REGION Network 17: AGAIN OFF TIME START AFTER RECIRCULATION OVER
   RUNG wire#powerrail
      Contact( "AlwaysTRUE" )
      { S7_Templates := "SrcType := Int" } EQ_Contact(in1 := "MODE SELECTION DB"."RO-2"."MODE BUFF", in2 := 1)
      { S7_Templates := "SrcType := Int" } EQ_Contact(in1 := "MODE SELECTION DB"."RO-2"."PROCESS BUFF", in2 := 2)
      { S7_Templates := "SrcType := Int" } EQ_Contact(in1 := "RO_2_LEVEL DB"."LEVEL HI RECIRC BUFF", in2 := 3)
      Contact( "TIMING_MIN_DB_10".DONE )
      Move(in := 4, out1 => "RO_2_LEVEL DB"."LEVEL HI RECIRC BUFF")
   END_RUNG
   // the same network as SCL:
   IF "AlwaysTRUE" AND ("MODE SELECTION DB"."RO-2"."MODE BUFF" = 1) AND ("MODE SELECTION DB"."RO-2"."PROCESS BUFF" = 2) AND ("RO_2_LEVEL DB"."LEVEL HI RECIRC BUFF" = 3) AND "TIMING_MIN_DB_10".DONE THEN
       "RO_2_LEVEL DB"."LEVEL HI RECIRC BUFF" := 4;
   END_IF;
END_REGION

REGION Network 18: AGAIN OFF TIME START AFTER RECIRCULATION OVER
   RUNG wire#powerrail
      Contact( "AlwaysTRUE" )
      { S7_Templates := "SrcType := Int" } EQ_Contact(in1 := "MODE SELECTION DB"."RO-2"."MODE BUFF", in2 := 1)
      { S7_Templates := "SrcType := Int" } EQ_Contact(in1 := "MODE SELECTION DB"."RO-2"."PROCESS BUFF", in2 := 2)
      { S7_Templates := "SrcType := Int" } EQ_Contact(in1 := "RO_2_LEVEL DB"."LEVEL HI RECIRC BUFF", in2 := 4)
      { S7_Templates := "time_type := Time" } "IEC_Timer_0_DB_95".TP(pt := T#2S, et =>)
      Move(in := 2, out1 => "RO_2_LEVEL DB"."LEVEL HI RECIRC BUFF")
   END_RUNG
   // the same network as SCL:
   "IEC_Timer_0_DB_95".TP(IN := "AlwaysTRUE" AND ("MODE SELECTION DB"."RO-2"."MODE BUFF" = 1) AND ("MODE SELECTION DB"."RO-2"."PROCESS BUFF" = 2) AND ("RO_2_LEVEL DB"."LEVEL HI RECIRC BUFF" = 4),
                          PT := T#2S);
   IF "IEC_Timer_0_DB_95".Q THEN "RO_2_LEVEL DB"."LEVEL HI RECIRC BUFF" := 2; END_IF;
END_REGION

REGION Network 19: REcirculation stop when level is normal
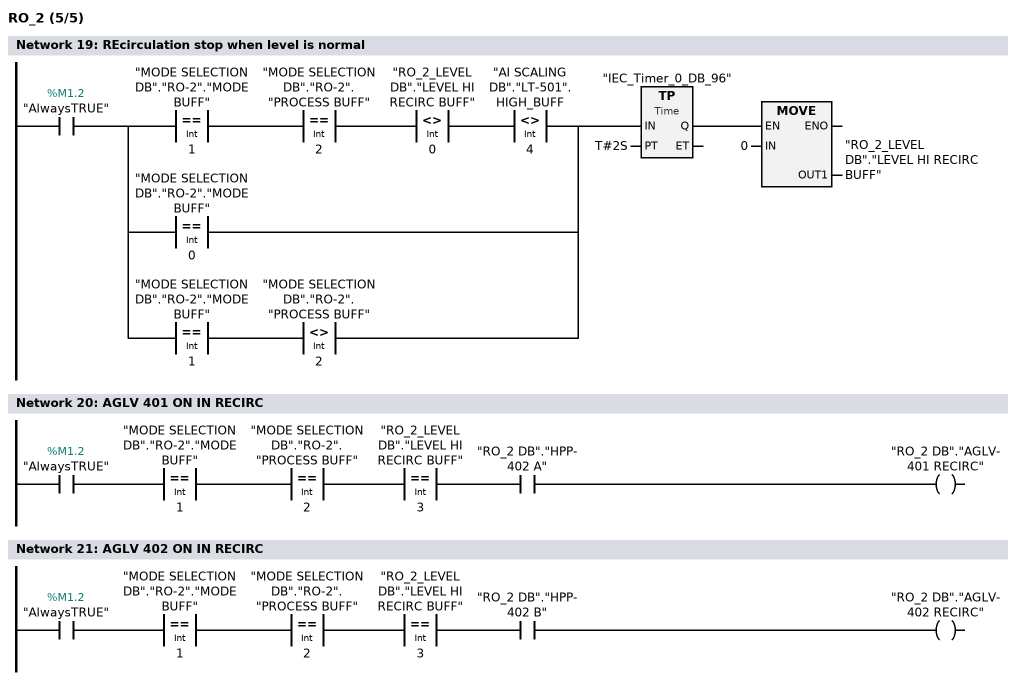
   RUNG wire#powerrail
      Contact( "AlwaysTRUE" )
      wire#w1
      { S7_Templates := "SrcType := Int" } EQ_Contact(in1 := "MODE SELECTION DB"."RO-2"."MODE BUFF", in2 := 1)
      { S7_Templates := "SrcType := Int" } EQ_Contact(in1 := "MODE SELECTION DB"."RO-2"."PROCESS BUFF", in2 := 2)
      { S7_Templates := "SrcType := Int" } NE_Contact(in1 := "RO_2_LEVEL DB"."LEVEL HI RECIRC BUFF", in2 := 0)
      { S7_Templates := "SrcType := Int" } NE_Contact(in1 := "AI SCALING DB"."LT-501".HIGH_BUFF, in2 := 4)
      wire#w2
      { S7_Templates := "time_type := Time" } "IEC_Timer_0_DB_96".TP(pt := T#2S, et =>)
      Move(in := 0, out1 => "RO_2_LEVEL DB"."LEVEL HI RECIRC BUFF")
   END_RUNG
   RUNG wire#w1
      { S7_Templates := "SrcType := Int" } EQ_Contact(in1 := "MODE SELECTION DB"."RO-2"."MODE BUFF", in2 := 0)
   END_RUNG wire#w2
   RUNG wire#w1
      { S7_Templates := "SrcType := Int" } EQ_Contact(in1 := "MODE SELECTION DB"."RO-2"."MODE BUFF", in2 := 1)
      { S7_Templates := "SrcType := Int" } NE_Contact(in1 := "MODE SELECTION DB"."RO-2"."PROCESS BUFF", in2 := 2)
   END_RUNG wire#w2
   // the same network as SCL:
   "IEC_Timer_0_DB_96".TP(IN := "AlwaysTRUE" AND ((("MODE SELECTION DB"."RO-2"."MODE BUFF" = 1) AND ("MODE SELECTION DB"."RO-2"."PROCESS BUFF" = 2) AND ("RO_2_LEVEL DB"."LEVEL HI RECIRC BUFF" <> 0) AND ("AI SCALING DB"."LT-501".HIGH_BUFF <> 4)) OR ("MODE SELECTION DB"."RO-2"."MODE BUFF" = 0) OR (("MODE SELECTION DB"."RO-2"."MODE BUFF" = 1) AND ("MODE SELECTION DB"."RO-2"."PROCESS BUFF" <> 2))),
                          PT := T#2S);
   IF "IEC_Timer_0_DB_96".Q THEN "RO_2_LEVEL DB"."LEVEL HI RECIRC BUFF" := 0; END_IF;
END_REGION

REGION Network 20: AGLV 401 ON IN RECIRC
   RUNG wire#powerrail
      Contact( "AlwaysTRUE" )
      { S7_Templates := "SrcType := Int" } EQ_Contact(in1 := "MODE SELECTION DB"."RO-2"."MODE BUFF", in2 := 1)
      { S7_Templates := "SrcType := Int" } EQ_Contact(in1 := "MODE SELECTION DB"."RO-2"."PROCESS BUFF", in2 := 2)
      { S7_Templates := "SrcType := Int" } EQ_Contact(in1 := "RO_2_LEVEL DB"."LEVEL HI RECIRC BUFF", in2 := 3)
      Contact( "RO_2 DB"."HPP-402 A" )
      Coil( "RO_2 DB"."AGLV-401 RECIRC" )
   END_RUNG
   // the same network as SCL:
   "RO_2 DB"."AGLV-401 RECIRC" := "AlwaysTRUE" AND ("MODE SELECTION DB"."RO-2"."MODE BUFF" = 1) AND ("MODE SELECTION DB"."RO-2"."PROCESS BUFF" = 2) AND ("RO_2_LEVEL DB"."LEVEL HI RECIRC BUFF" = 3) AND "RO_2 DB"."HPP-402 A";
END_REGION

REGION Network 21: AGLV 402 ON IN RECIRC
   RUNG wire#powerrail
      Contact( "AlwaysTRUE" )
      { S7_Templates := "SrcType := Int" } EQ_Contact(in1 := "MODE SELECTION DB"."RO-2"."MODE BUFF", in2 := 1)
      { S7_Templates := "SrcType := Int" } EQ_Contact(in1 := "MODE SELECTION DB"."RO-2"."PROCESS BUFF", in2 := 2)
      { S7_Templates := "SrcType := Int" } EQ_Contact(in1 := "RO_2_LEVEL DB"."LEVEL HI RECIRC BUFF", in2 := 3)
      Contact( "RO_2 DB"."HPP-402 B" )
      Coil( "RO_2 DB"."AGLV-402 RECIRC" )
   END_RUNG
   // the same network as SCL:
   "RO_2 DB"."AGLV-402 RECIRC" := "AlwaysTRUE" AND ("MODE SELECTION DB"."RO-2"."MODE BUFF" = 1) AND ("MODE SELECTION DB"."RO-2"."PROCESS BUFF" = 2) AND ("RO_2_LEVEL DB"."LEVEL HI RECIRC BUFF" = 3) AND "RO_2 DB"."HPP-402 B";
END_REGION
END_FUNCTION

FUNCTION "EDI" : Void   // FC12, LAD
{ S7_Optimized_Access := 'TRUE' }
// stored: SetENOAutomatically false
   VAR_TEMP   // added for the SCL form of the ladder/FBD networks
      _w1 : Bool;
   END_VAR
BEGIN

REGION Network 1: FEED PUMP
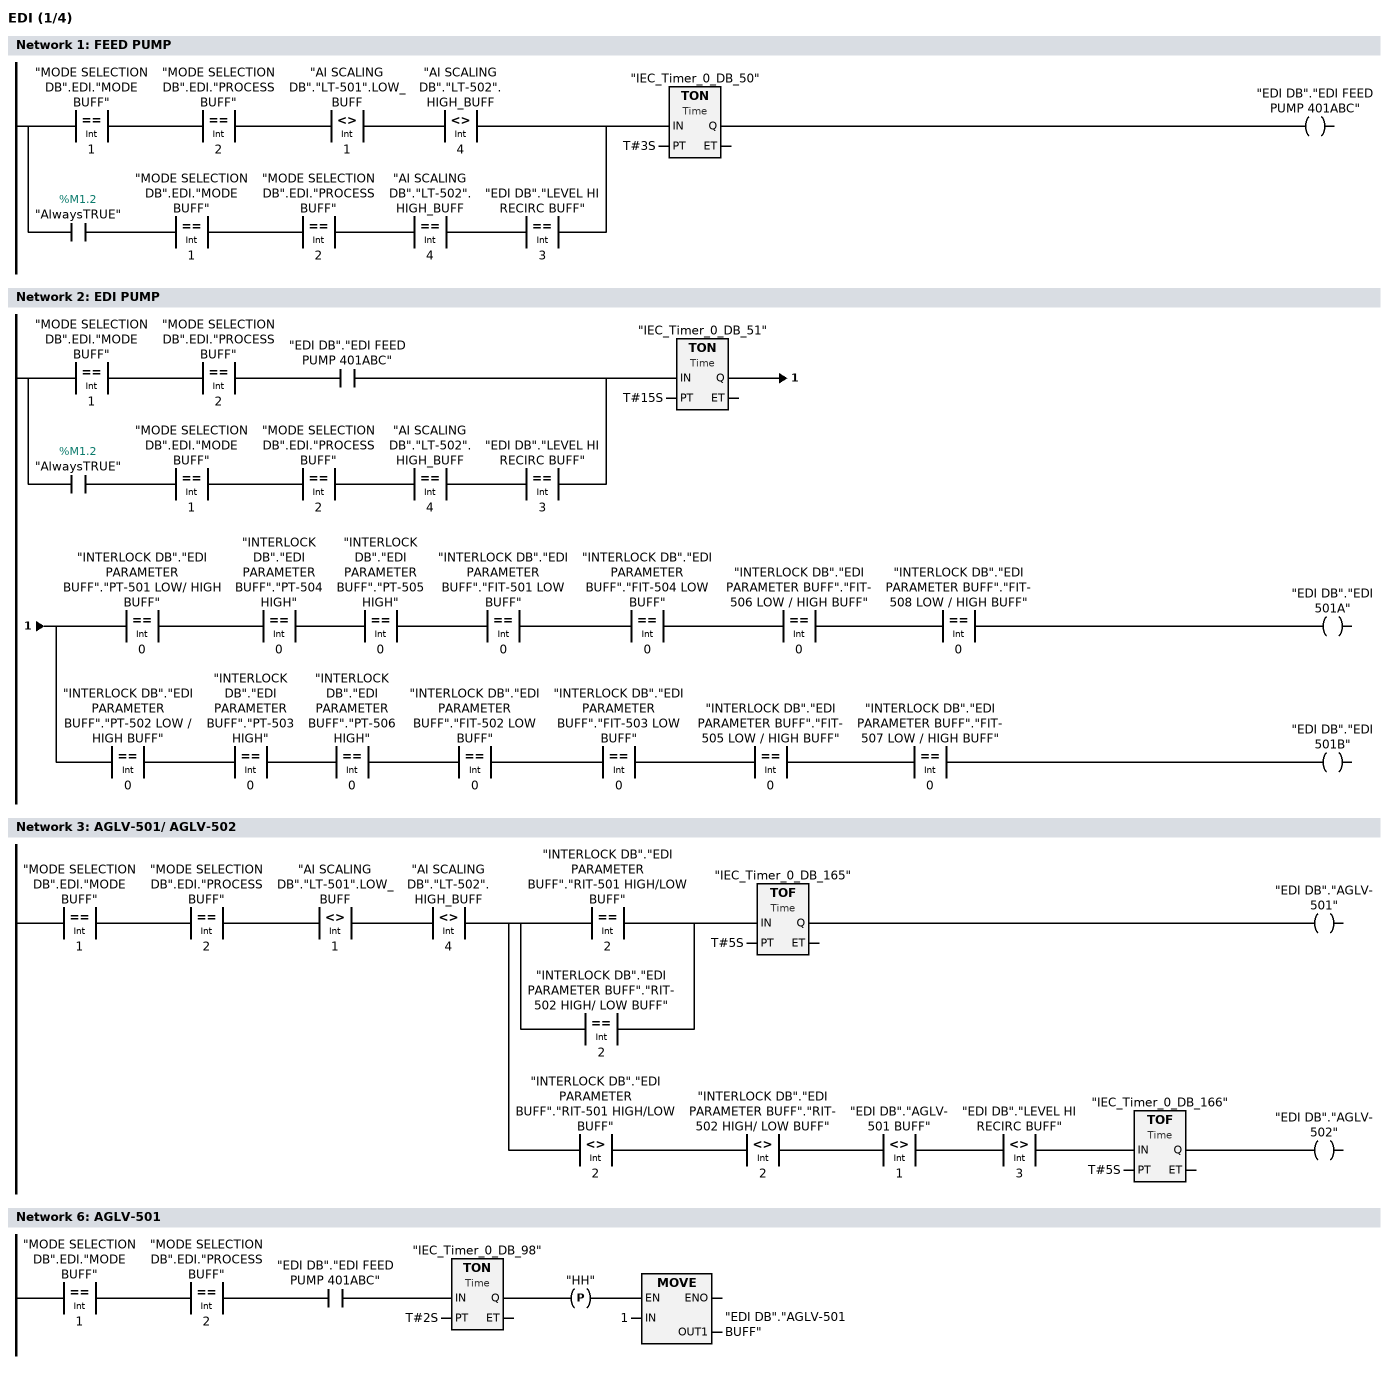
   RUNG wire#powerrail
      { S7_Templates := "SrcType := Int" } EQ_Contact(in1 := "MODE SELECTION DB".EDI."MODE BUFF", in2 := 1)
      { S7_Templates := "SrcType := Int" } EQ_Contact(in1 := "MODE SELECTION DB".EDI."PROCESS BUFF", in2 := 2)
      { S7_Templates := "SrcType := Int" } NE_Contact(in1 := "AI SCALING DB"."LT-501".LOW_BUFF, in2 := 1)
      { S7_Templates := "SrcType := Int" } NE_Contact(in1 := "AI SCALING DB"."LT-502".HIGH_BUFF, in2 := 4)
      wire#w1
      { S7_Templates := "time_type := Time" } "IEC_Timer_0_DB_50".TON(pt := T#3S, et =>)
      Coil( "EDI DB"."EDI FEED PUMP 401ABC" )
   END_RUNG
   RUNG wire#powerrail
      Contact( "AlwaysTRUE" )
      { S7_Templates := "SrcType := Int" } EQ_Contact(in1 := "MODE SELECTION DB".EDI."MODE BUFF", in2 := 1)
      { S7_Templates := "SrcType := Int" } EQ_Contact(in1 := "MODE SELECTION DB".EDI."PROCESS BUFF", in2 := 2)
      { S7_Templates := "SrcType := Int" } EQ_Contact(in1 := "AI SCALING DB"."LT-502".HIGH_BUFF, in2 := 4)
      { S7_Templates := "SrcType := Int" } EQ_Contact(in1 := "EDI DB"."LEVEL HI RECIRC BUFF", in2 := 3)
   END_RUNG wire#w1
   // the same network as SCL:
   "IEC_Timer_0_DB_50".TON(IN := (("MODE SELECTION DB".EDI."MODE BUFF" = 1) AND ("MODE SELECTION DB".EDI."PROCESS BUFF" = 2) AND ("AI SCALING DB"."LT-501".LOW_BUFF <> 1) AND ("AI SCALING DB"."LT-502".HIGH_BUFF <> 4)) OR ("AlwaysTRUE" AND ("MODE SELECTION DB".EDI."MODE BUFF" = 1) AND ("MODE SELECTION DB".EDI."PROCESS BUFF" = 2) AND ("AI SCALING DB"."LT-502".HIGH_BUFF = 4) AND ("EDI DB"."LEVEL HI RECIRC BUFF" = 3)),
                           PT := T#3S);
   "EDI DB"."EDI FEED PUMP 401ABC" := "IEC_Timer_0_DB_50".Q;
END_REGION

REGION Network 2: EDI PUMP
   RUNG wire#powerrail
      { S7_Templates := "SrcType := Int" } EQ_Contact(in1 := "MODE SELECTION DB".EDI."MODE BUFF", in2 := 1)
      { S7_Templates := "SrcType := Int" } EQ_Contact(in1 := "MODE SELECTION DB".EDI."PROCESS BUFF", in2 := 2)
      Contact( "EDI DB"."EDI FEED PUMP 401ABC" )
      wire#w1
      { S7_Templates := "time_type := Time" } "IEC_Timer_0_DB_51".TON(pt := T#15S, et =>)
      wire#w2
      { S7_Templates := "SrcType := Int" } EQ_Contact(in1 := "INTERLOCK DB"."EDI PARAMETER BUFF"."PT-501 LOW/ HIGH BUFF", in2 := 0)
      { S7_Templates := "SrcType := Int" } EQ_Contact(in1 := "INTERLOCK DB"."EDI PARAMETER BUFF"."PT-504 HIGH", in2 := 0)
      { S7_Templates := "SrcType := Int" } EQ_Contact(in1 := "INTERLOCK DB"."EDI PARAMETER BUFF"."PT-505 HIGH", in2 := 0)
      { S7_Templates := "SrcType := Int" } EQ_Contact(in1 := "INTERLOCK DB"."EDI PARAMETER BUFF"."FIT-501 LOW BUFF", in2 := 0)
      { S7_Templates := "SrcType := Int" } EQ_Contact(in1 := "INTERLOCK DB"."EDI PARAMETER BUFF"."FIT-504 LOW BUFF", in2 := 0)
      { S7_Templates := "SrcType := Int" } EQ_Contact(in1 := "INTERLOCK DB"."EDI PARAMETER BUFF"."FIT-506 LOW / HIGH BUFF", in2 := 0)
      { S7_Templates := "SrcType := Int" } EQ_Contact(in1 := "INTERLOCK DB"."EDI PARAMETER BUFF"."FIT-508 LOW / HIGH BUFF", in2 := 0)
      Coil( "EDI DB"."EDI 501A" )
   END_RUNG
   RUNG wire#powerrail
      Contact( "AlwaysTRUE" )
      { S7_Templates := "SrcType := Int" } EQ_Contact(in1 := "MODE SELECTION DB".EDI."MODE BUFF", in2 := 1)
      { S7_Templates := "SrcType := Int" } EQ_Contact(in1 := "MODE SELECTION DB".EDI."PROCESS BUFF", in2 := 2)
      { S7_Templates := "SrcType := Int" } EQ_Contact(in1 := "AI SCALING DB"."LT-502".HIGH_BUFF, in2 := 4)
      { S7_Templates := "SrcType := Int" } EQ_Contact(in1 := "EDI DB"."LEVEL HI RECIRC BUFF", in2 := 3)
   END_RUNG wire#w1
   RUNG wire#w2
      { S7_Templates := "SrcType := Int" } EQ_Contact(in1 := "INTERLOCK DB"."EDI PARAMETER BUFF"."PT-502 LOW / HIGH BUFF", in2 := 0)
      { S7_Templates := "SrcType := Int" } EQ_Contact(in1 := "INTERLOCK DB"."EDI PARAMETER BUFF"."PT-503 HIGH", in2 := 0)
      { S7_Templates := "SrcType := Int" } EQ_Contact(in1 := "INTERLOCK DB"."EDI PARAMETER BUFF"."PT-506 HIGH", in2 := 0)
      { S7_Templates := "SrcType := Int" } EQ_Contact(in1 := "INTERLOCK DB"."EDI PARAMETER BUFF"."FIT-502 LOW  BUFF", in2 := 0)
      { S7_Templates := "SrcType := Int" } EQ_Contact(in1 := "INTERLOCK DB"."EDI PARAMETER BUFF"."FIT-503 LOW BUFF", in2 := 0)
      { S7_Templates := "SrcType := Int" } EQ_Contact(in1 := "INTERLOCK DB"."EDI PARAMETER BUFF"."FIT-505 LOW / HIGH BUFF", in2 := 0)
      { S7_Templates := "SrcType := Int" } EQ_Contact(in1 := "INTERLOCK DB"."EDI PARAMETER BUFF"."FIT-507 LOW / HIGH BUFF", in2 := 0)
      Coil( "EDI DB"."EDI 501B" )
   END_RUNG
   // the same network as SCL:
   "IEC_Timer_0_DB_51".TON(IN := (("MODE SELECTION DB".EDI."MODE BUFF" = 1) AND ("MODE SELECTION DB".EDI."PROCESS BUFF" = 2) AND "EDI DB"."EDI FEED PUMP 401ABC") OR ("AlwaysTRUE" AND ("MODE SELECTION DB".EDI."MODE BUFF" = 1) AND ("MODE SELECTION DB".EDI."PROCESS BUFF" = 2) AND ("AI SCALING DB"."LT-502".HIGH_BUFF = 4) AND ("EDI DB"."LEVEL HI RECIRC BUFF" = 3)),
                           PT := T#15S);
   "EDI DB"."EDI 501A" := "IEC_Timer_0_DB_51".Q AND ("INTERLOCK DB"."EDI PARAMETER BUFF"."PT-501 LOW/ HIGH BUFF" = 0) AND ("INTERLOCK DB"."EDI PARAMETER BUFF"."PT-504 HIGH" = 0) AND ("INTERLOCK DB"."EDI PARAMETER BUFF"."PT-505 HIGH" = 0) AND ("INTERLOCK DB"."EDI PARAMETER BUFF"."FIT-501 LOW BUFF" = 0) AND ("INTERLOCK DB"."EDI PARAMETER BUFF"."FIT-504 LOW BUFF" = 0) AND ("INTERLOCK DB"."EDI PARAMETER BUFF"."FIT-506 LOW / HIGH BUFF" = 0) AND ("INTERLOCK DB"."EDI PARAMETER BUFF"."FIT-508 LOW / HIGH BUFF" = 0);
   "EDI DB"."EDI 501B" := "IEC_Timer_0_DB_51".Q AND ("INTERLOCK DB"."EDI PARAMETER BUFF"."PT-502 LOW / HIGH BUFF" = 0) AND ("INTERLOCK DB"."EDI PARAMETER BUFF"."PT-503 HIGH" = 0) AND ("INTERLOCK DB"."EDI PARAMETER BUFF"."PT-506 HIGH" = 0) AND ("INTERLOCK DB"."EDI PARAMETER BUFF"."FIT-502 LOW  BUFF" = 0) AND ("INTERLOCK DB"."EDI PARAMETER BUFF"."FIT-503 LOW BUFF" = 0) AND ("INTERLOCK DB"."EDI PARAMETER BUFF"."FIT-505 LOW / HIGH BUFF" = 0) AND ("INTERLOCK DB"."EDI PARAMETER BUFF"."FIT-507 LOW / HIGH BUFF" = 0);
END_REGION

REGION Network 3: AGLV-501/ AGLV-502
   RUNG wire#powerrail
      { S7_Templates := "SrcType := Int" } EQ_Contact(in1 := "MODE SELECTION DB".EDI."MODE BUFF", in2 := 1)
      { S7_Templates := "SrcType := Int" } EQ_Contact(in1 := "MODE SELECTION DB".EDI."PROCESS BUFF", in2 := 2)
      { S7_Templates := "SrcType := Int" } NE_Contact(in1 := "AI SCALING DB"."LT-501".LOW_BUFF, in2 := 1)
      { S7_Templates := "SrcType := Int" } NE_Contact(in1 := "AI SCALING DB"."LT-502".HIGH_BUFF, in2 := 4)
      wire#w1
      { S7_Templates := "SrcType := Int" } EQ_Contact(in1 := "INTERLOCK DB"."EDI PARAMETER BUFF"."RIT-501 HIGH/LOW BUFF", in2 := 2)
      wire#w2
      { S7_Templates := "time_type := Time" } "IEC_Timer_0_DB_165".TOF(pt := T#5S, et =>)
      Coil( "EDI DB"."AGLV-501" )
   END_RUNG
   RUNG wire#w1
      { S7_Templates := "SrcType := Int" } EQ_Contact(in1 := "INTERLOCK DB"."EDI PARAMETER BUFF"."RIT-502 HIGH/ LOW BUFF", in2 := 2)
   END_RUNG wire#w2
   RUNG wire#w1
      { S7_Templates := "SrcType := Int" } NE_Contact(in1 := "INTERLOCK DB"."EDI PARAMETER BUFF"."RIT-501 HIGH/LOW BUFF", in2 := 2)
      { S7_Templates := "SrcType := Int" } NE_Contact(in1 := "INTERLOCK DB"."EDI PARAMETER BUFF"."RIT-502 HIGH/ LOW BUFF", in2 := 2)
      { S7_Templates := "SrcType := Int" } NE_Contact(in1 := "EDI DB"."AGLV-501 BUFF", in2 := 1)
      { S7_Templates := "SrcType := Int" } NE_Contact(in1 := "EDI DB"."LEVEL HI RECIRC BUFF", in2 := 3)
      { S7_Templates := "time_type := Time" } "IEC_Timer_0_DB_166".TOF(pt := T#5S, et =>)
      Coil( "EDI DB"."AGLV-502" )
   END_RUNG
   // the same network as SCL:
   #_w1 := ("MODE SELECTION DB".EDI."MODE BUFF" = 1) AND ("MODE SELECTION DB".EDI."PROCESS BUFF" = 2) AND ("AI SCALING DB"."LT-501".LOW_BUFF <> 1) AND ("AI SCALING DB"."LT-502".HIGH_BUFF <> 4);
   "IEC_Timer_0_DB_165".TOF(IN := #_w1 AND (("INTERLOCK DB"."EDI PARAMETER BUFF"."RIT-501 HIGH/LOW BUFF" = 2) OR ("INTERLOCK DB"."EDI PARAMETER BUFF"."RIT-502 HIGH/ LOW BUFF" = 2)),
                           PT := T#5S);
   "EDI DB"."AGLV-501" := "IEC_Timer_0_DB_165".Q;
   "IEC_Timer_0_DB_166".TOF(IN := #_w1 AND ("INTERLOCK DB"."EDI PARAMETER BUFF"."RIT-501 HIGH/LOW BUFF" <> 2) AND ("INTERLOCK DB"."EDI PARAMETER BUFF"."RIT-502 HIGH/ LOW BUFF" <> 2) AND ("EDI DB"."AGLV-501 BUFF" <> 1) AND ("EDI DB"."LEVEL HI RECIRC BUFF" <> 3),
                           PT := T#5S);
   "EDI DB"."AGLV-502" := "IEC_Timer_0_DB_166".Q;
END_REGION

REGION Network 6: AGLV-501
   RUNG wire#powerrail
      { S7_Templates := "SrcType := Int" } EQ_Contact(in1 := "MODE SELECTION DB".EDI."MODE BUFF", in2 := 1)
      { S7_Templates := "SrcType := Int" } EQ_Contact(in1 := "MODE SELECTION DB".EDI."PROCESS BUFF", in2 := 2)
      Contact( "EDI DB"."EDI FEED PUMP 401ABC" )
      { S7_Templates := "time_type := Time" } "IEC_Timer_0_DB_98".TON(pt := T#2S, et =>)
      P_Trig( "HH" )
      Move(in := 1, out1 => "EDI DB"."AGLV-501 BUFF")
   END_RUNG
   // the same network as SCL:
   "IEC_Timer_0_DB_98".TON(IN := ("MODE SELECTION DB".EDI."MODE BUFF" = 1) AND ("MODE SELECTION DB".EDI."PROCESS BUFF" = 2) AND "EDI DB"."EDI FEED PUMP 401ABC",
                           PT := T#2S);
   #_w1 := "IEC_Timer_0_DB_98".Q AND NOT "HH";   // rising edge
   "HH" := "IEC_Timer_0_DB_98".Q;
   IF #_w1 THEN "EDI DB"."AGLV-501 BUFF" := 1; END_IF;
END_REGION

REGION Network 7
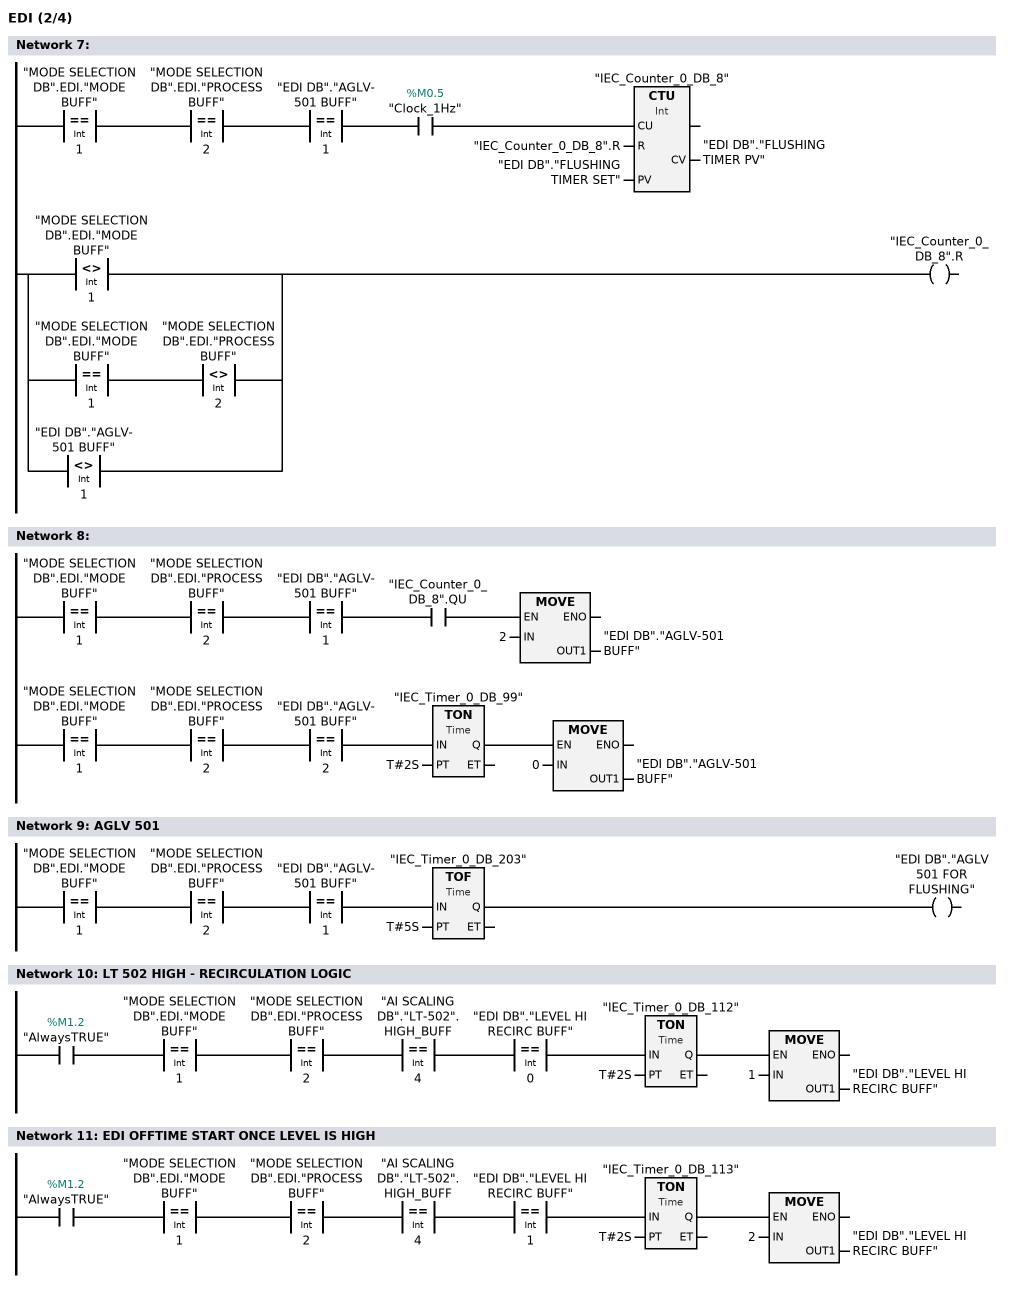
   RUNG wire#powerrail
      { S7_Templates := "SrcType := Int" } EQ_Contact(in1 := "MODE SELECTION DB".EDI."MODE BUFF", in2 := 1)
      { S7_Templates := "SrcType := Int" } EQ_Contact(in1 := "MODE SELECTION DB".EDI."PROCESS BUFF", in2 := 2)
      { S7_Templates := "SrcType := Int" } EQ_Contact(in1 := "EDI DB"."AGLV-501 BUFF", in2 := 1)
      Contact( "Clock_1Hz" )
      { S7_Templates := "value_type := Int" } "IEC_Counter_0_DB_8".CTU(r := "IEC_Counter_0_DB_8".R, pv := "EDI DB"."FLUSHING TIMER SET", cv => "EDI DB"."FLUSHING TIMER PV")
   END_RUNG
   RUNG wire#powerrail
      { S7_Templates := "SrcType := Int" } NE_Contact(in1 := "MODE SELECTION DB".EDI."MODE BUFF", in2 := 1)
      wire#w1
      Coil( "IEC_Counter_0_DB_8".R )
   END_RUNG
   RUNG wire#powerrail
      { S7_Templates := "SrcType := Int" } EQ_Contact(in1 := "MODE SELECTION DB".EDI."MODE BUFF", in2 := 1)
      { S7_Templates := "SrcType := Int" } NE_Contact(in1 := "MODE SELECTION DB".EDI."PROCESS BUFF", in2 := 2)
   END_RUNG wire#w1
   RUNG wire#powerrail
      { S7_Templates := "SrcType := Int" } NE_Contact(in1 := "EDI DB"."AGLV-501 BUFF", in2 := 1)
   END_RUNG wire#w1
   // the same network as SCL:
   "IEC_Counter_0_DB_8".CTU(CU := ("MODE SELECTION DB".EDI."MODE BUFF" = 1) AND ("MODE SELECTION DB".EDI."PROCESS BUFF" = 2) AND ("EDI DB"."AGLV-501 BUFF" = 1) AND "Clock_1Hz",
                           R := "IEC_Counter_0_DB_8".R,
                           PV := "EDI DB"."FLUSHING TIMER SET",
                           CV => "EDI DB"."FLUSHING TIMER PV");
   "IEC_Counter_0_DB_8".R := ("MODE SELECTION DB".EDI."MODE BUFF" <> 1) OR (("MODE SELECTION DB".EDI."MODE BUFF" = 1) AND ("MODE SELECTION DB".EDI."PROCESS BUFF" <> 2)) OR ("EDI DB"."AGLV-501 BUFF" <> 1);
END_REGION

REGION Network 8
   RUNG wire#powerrail
      { S7_Templates := "SrcType := Int" } EQ_Contact(in1 := "MODE SELECTION DB".EDI."MODE BUFF", in2 := 1)
      { S7_Templates := "SrcType := Int" } EQ_Contact(in1 := "MODE SELECTION DB".EDI."PROCESS BUFF", in2 := 2)
      { S7_Templates := "SrcType := Int" } EQ_Contact(in1 := "EDI DB"."AGLV-501 BUFF", in2 := 1)
      Contact( "IEC_Counter_0_DB_8".QU )
      Move(in := 2, out1 => "EDI DB"."AGLV-501 BUFF")
   END_RUNG
   RUNG wire#powerrail
      { S7_Templates := "SrcType := Int" } EQ_Contact(in1 := "MODE SELECTION DB".EDI."MODE BUFF", in2 := 1)
      { S7_Templates := "SrcType := Int" } EQ_Contact(in1 := "MODE SELECTION DB".EDI."PROCESS BUFF", in2 := 2)
      { S7_Templates := "SrcType := Int" } EQ_Contact(in1 := "EDI DB"."AGLV-501 BUFF", in2 := 2)
      { S7_Templates := "time_type := Time" } "IEC_Timer_0_DB_99".TON(pt := T#2S, et =>)
      Move(in := 0, out1 => "EDI DB"."AGLV-501 BUFF")
   END_RUNG
   // the same network as SCL:
   IF ("MODE SELECTION DB".EDI."MODE BUFF" = 1) AND ("MODE SELECTION DB".EDI."PROCESS BUFF" = 2) AND ("EDI DB"."AGLV-501 BUFF" = 1) AND "IEC_Counter_0_DB_8".QU THEN
       "EDI DB"."AGLV-501 BUFF" := 2;
   END_IF;
   "IEC_Timer_0_DB_99".TON(IN := ("MODE SELECTION DB".EDI."MODE BUFF" = 1) AND ("MODE SELECTION DB".EDI."PROCESS BUFF" = 2) AND ("EDI DB"."AGLV-501 BUFF" = 2),
                           PT := T#2S);
   IF "IEC_Timer_0_DB_99".Q THEN "EDI DB"."AGLV-501 BUFF" := 0; END_IF;
END_REGION

REGION Network 9: AGLV 501
   RUNG wire#powerrail
      { S7_Templates := "SrcType := Int" } EQ_Contact(in1 := "MODE SELECTION DB".EDI."MODE BUFF", in2 := 1)
      { S7_Templates := "SrcType := Int" } EQ_Contact(in1 := "MODE SELECTION DB".EDI."PROCESS BUFF", in2 := 2)
      { S7_Templates := "SrcType := Int" } EQ_Contact(in1 := "EDI DB"."AGLV-501 BUFF", in2 := 1)
      { S7_Templates := "time_type := Time" } "IEC_Timer_0_DB_203".TOF(pt := T#5S, et =>)
      Coil( "EDI DB"."AGLV 501 FOR FLUSHING" )
   END_RUNG
   // the same network as SCL:
   "IEC_Timer_0_DB_203".TOF(IN := ("MODE SELECTION DB".EDI."MODE BUFF" = 1) AND ("MODE SELECTION DB".EDI."PROCESS BUFF" = 2) AND ("EDI DB"."AGLV-501 BUFF" = 1),
                           PT := T#5S);
   "EDI DB"."AGLV 501 FOR FLUSHING" := "IEC_Timer_0_DB_203".Q;
END_REGION

REGION Network 10: LT 502 HIGH - RECIRCULATION LOGIC
   RUNG wire#powerrail
      Contact( "AlwaysTRUE" )
      { S7_Templates := "SrcType := Int" } EQ_Contact(in1 := "MODE SELECTION DB".EDI."MODE BUFF", in2 := 1)
      { S7_Templates := "SrcType := Int" } EQ_Contact(in1 := "MODE SELECTION DB".EDI."PROCESS BUFF", in2 := 2)
      { S7_Templates := "SrcType := Int" } EQ_Contact(in1 := "AI SCALING DB"."LT-502".HIGH_BUFF, in2 := 4)
      { S7_Templates := "SrcType := Int" } EQ_Contact(in1 := "EDI DB"."LEVEL HI RECIRC BUFF", in2 := 0)
      { S7_Templates := "time_type := Time" } "IEC_Timer_0_DB_112".TON(pt := T#2S, et =>)
      Move(in := 1, out1 => "EDI DB"."LEVEL HI RECIRC BUFF")
   END_RUNG
   // the same network as SCL:
   "IEC_Timer_0_DB_112".TON(IN := "AlwaysTRUE" AND ("MODE SELECTION DB".EDI."MODE BUFF" = 1) AND ("MODE SELECTION DB".EDI."PROCESS BUFF" = 2) AND ("AI SCALING DB"."LT-502".HIGH_BUFF = 4) AND ("EDI DB"."LEVEL HI RECIRC BUFF" = 0),
                           PT := T#2S);
   IF "IEC_Timer_0_DB_112".Q THEN "EDI DB"."LEVEL HI RECIRC BUFF" := 1; END_IF;
END_REGION

REGION Network 11: EDI OFFTIME START ONCE LEVEL IS HIGH
   RUNG wire#powerrail
      Contact( "AlwaysTRUE" )
      { S7_Templates := "SrcType := Int" } EQ_Contact(in1 := "MODE SELECTION DB".EDI."MODE BUFF", in2 := 1)
      { S7_Templates := "SrcType := Int" } EQ_Contact(in1 := "MODE SELECTION DB".EDI."PROCESS BUFF", in2 := 2)
      { S7_Templates := "SrcType := Int" } EQ_Contact(in1 := "AI SCALING DB"."LT-502".HIGH_BUFF, in2 := 4)
      { S7_Templates := "SrcType := Int" } EQ_Contact(in1 := "EDI DB"."LEVEL HI RECIRC BUFF", in2 := 1)
      { S7_Templates := "time_type := Time" } "IEC_Timer_0_DB_113".TON(pt := T#2S, et =>)
      Move(in := 2, out1 => "EDI DB"."LEVEL HI RECIRC BUFF")
   END_RUNG
   // the same network as SCL:
   "IEC_Timer_0_DB_113".TON(IN := "AlwaysTRUE" AND ("MODE SELECTION DB".EDI."MODE BUFF" = 1) AND ("MODE SELECTION DB".EDI."PROCESS BUFF" = 2) AND ("AI SCALING DB"."LT-502".HIGH_BUFF = 4) AND ("EDI DB"."LEVEL HI RECIRC BUFF" = 1),
                           PT := T#2S);
   IF "IEC_Timer_0_DB_113".Q THEN "EDI DB"."LEVEL HI RECIRC BUFF" := 2; END_IF;
END_REGION

REGION Network 12: EDI OFF TIME START
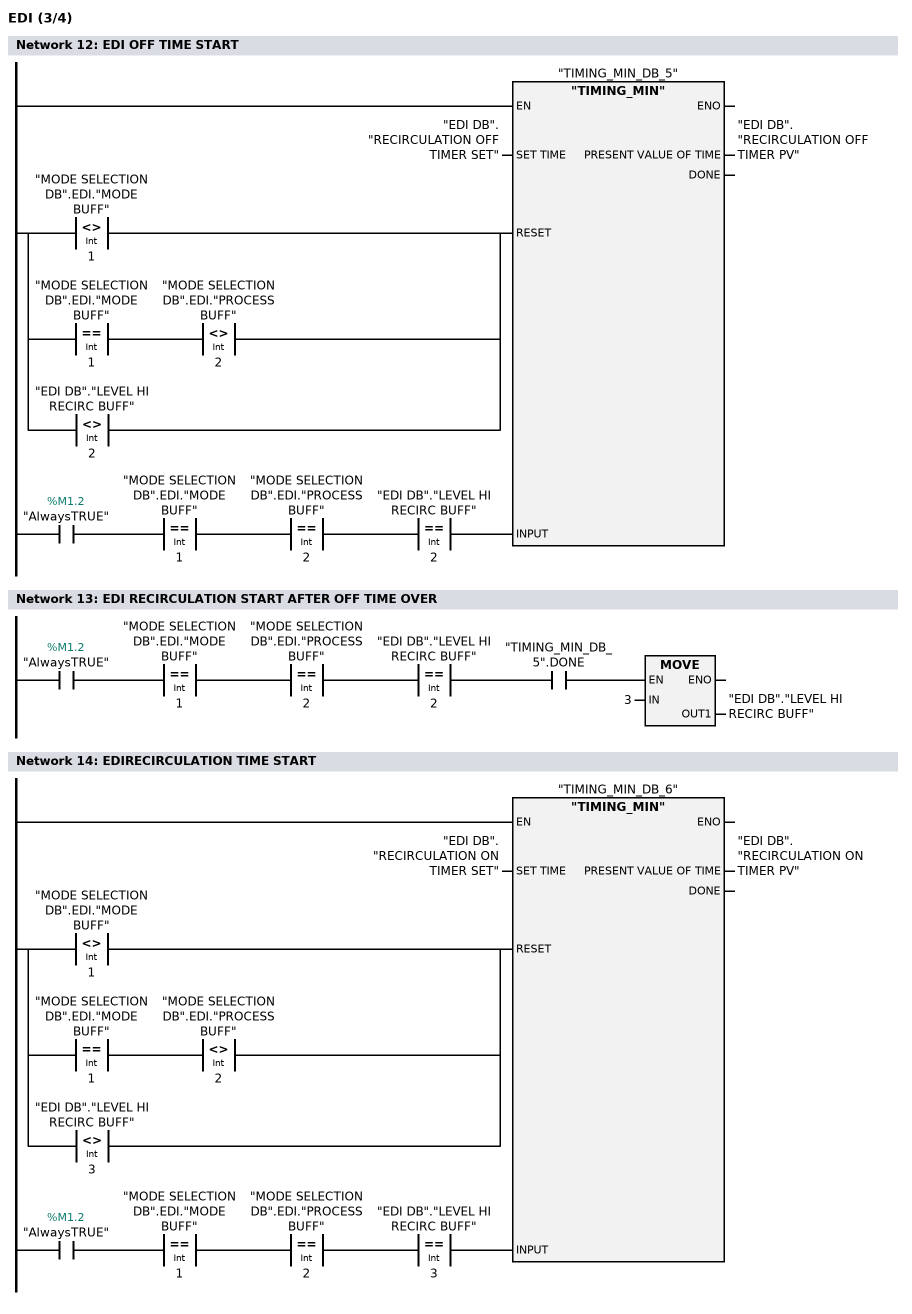
   RUNG wire#powerrail
      "TIMING_MIN_DB_5"(RESET := wire#w1, INPUT := wire#w2, "SET TIME" := "EDI DB"."RECIRCULATION OFF TIMER SET", "PRESENT VALUE OF TIME" => "EDI DB"."RECIRCULATION OFF TIMER PV", DONE =>)
   END_RUNG
   RUNG wire#powerrail
      { S7_Templates := "SrcType := Int" } NE_Contact(in1 := "MODE SELECTION DB".EDI."MODE BUFF", in2 := 1)
   END_RUNG wire#w1
   RUNG wire#powerrail
      { S7_Templates := "SrcType := Int" } EQ_Contact(in1 := "MODE SELECTION DB".EDI."MODE BUFF", in2 := 1)
      { S7_Templates := "SrcType := Int" } NE_Contact(in1 := "MODE SELECTION DB".EDI."PROCESS BUFF", in2 := 2)
   END_RUNG wire#w1
   RUNG wire#powerrail
      { S7_Templates := "SrcType := Int" } NE_Contact(in1 := "EDI DB"."LEVEL HI RECIRC BUFF", in2 := 2)
   END_RUNG wire#w1
   RUNG wire#powerrail
      Contact( "AlwaysTRUE" )
      { S7_Templates := "SrcType := Int" } EQ_Contact(in1 := "MODE SELECTION DB".EDI."MODE BUFF", in2 := 1)
      { S7_Templates := "SrcType := Int" } EQ_Contact(in1 := "MODE SELECTION DB".EDI."PROCESS BUFF", in2 := 2)
      { S7_Templates := "SrcType := Int" } EQ_Contact(in1 := "EDI DB"."LEVEL HI RECIRC BUFF", in2 := 2)
   END_RUNG wire#w2
   // the same network as SCL:
   "TIMING_MIN_DB_5"("SET TIME" := "EDI DB"."RECIRCULATION OFF TIMER SET",   // "TIMING_MIN"
                     RESET := ("MODE SELECTION DB".EDI."MODE BUFF" <> 1) OR (("MODE SELECTION DB".EDI."MODE BUFF" = 1) AND ("MODE SELECTION DB".EDI."PROCESS BUFF" <> 2)) OR ("EDI DB"."LEVEL HI RECIRC BUFF" <> 2),
                     INPUT := "AlwaysTRUE" AND ("MODE SELECTION DB".EDI."MODE BUFF" = 1) AND ("MODE SELECTION DB".EDI."PROCESS BUFF" = 2) AND ("EDI DB"."LEVEL HI RECIRC BUFF" = 2),
                     "PRESENT VALUE OF TIME" => "EDI DB"."RECIRCULATION OFF TIMER PV");
END_REGION

REGION Network 13: EDI RECIRCULATION START AFTER OFF TIME OVER
   RUNG wire#powerrail
      Contact( "AlwaysTRUE" )
      { S7_Templates := "SrcType := Int" } EQ_Contact(in1 := "MODE SELECTION DB".EDI."MODE BUFF", in2 := 1)
      { S7_Templates := "SrcType := Int" } EQ_Contact(in1 := "MODE SELECTION DB".EDI."PROCESS BUFF", in2 := 2)
      { S7_Templates := "SrcType := Int" } EQ_Contact(in1 := "EDI DB"."LEVEL HI RECIRC BUFF", in2 := 2)
      Contact( "TIMING_MIN_DB_5".DONE )
      Move(in := 3, out1 => "EDI DB"."LEVEL HI RECIRC BUFF")
   END_RUNG
   // the same network as SCL:
   IF "AlwaysTRUE" AND ("MODE SELECTION DB".EDI."MODE BUFF" = 1) AND ("MODE SELECTION DB".EDI."PROCESS BUFF" = 2) AND ("EDI DB"."LEVEL HI RECIRC BUFF" = 2) AND "TIMING_MIN_DB_5".DONE THEN
       "EDI DB"."LEVEL HI RECIRC BUFF" := 3;
   END_IF;
END_REGION

REGION Network 14: EDIRECIRCULATION TIME START
   RUNG wire#powerrail
      "TIMING_MIN_DB_6"(RESET := wire#w1, INPUT := wire#w2, "SET TIME" := "EDI DB"."RECIRCULATION ON TIMER SET", "PRESENT VALUE OF TIME" => "EDI DB"."RECIRCULATION ON TIMER PV", DONE =>)
   END_RUNG
   RUNG wire#powerrail
      { S7_Templates := "SrcType := Int" } NE_Contact(in1 := "MODE SELECTION DB".EDI."MODE BUFF", in2 := 1)
   END_RUNG wire#w1
   RUNG wire#powerrail
      { S7_Templates := "SrcType := Int" } EQ_Contact(in1 := "MODE SELECTION DB".EDI."MODE BUFF", in2 := 1)
      { S7_Templates := "SrcType := Int" } NE_Contact(in1 := "MODE SELECTION DB".EDI."PROCESS BUFF", in2 := 2)
   END_RUNG wire#w1
   RUNG wire#powerrail
      { S7_Templates := "SrcType := Int" } NE_Contact(in1 := "EDI DB"."LEVEL HI RECIRC BUFF", in2 := 3)
   END_RUNG wire#w1
   RUNG wire#powerrail
      Contact( "AlwaysTRUE" )
      { S7_Templates := "SrcType := Int" } EQ_Contact(in1 := "MODE SELECTION DB".EDI."MODE BUFF", in2 := 1)
      { S7_Templates := "SrcType := Int" } EQ_Contact(in1 := "MODE SELECTION DB".EDI."PROCESS BUFF", in2 := 2)
      { S7_Templates := "SrcType := Int" } EQ_Contact(in1 := "EDI DB"."LEVEL HI RECIRC BUFF", in2 := 3)
   END_RUNG wire#w2
   // the same network as SCL:
   "TIMING_MIN_DB_6"("SET TIME" := "EDI DB"."RECIRCULATION ON TIMER SET",   // "TIMING_MIN"
                     RESET := ("MODE SELECTION DB".EDI."MODE BUFF" <> 1) OR (("MODE SELECTION DB".EDI."MODE BUFF" = 1) AND ("MODE SELECTION DB".EDI."PROCESS BUFF" <> 2)) OR ("EDI DB"."LEVEL HI RECIRC BUFF" <> 3),
                     INPUT := "AlwaysTRUE" AND ("MODE SELECTION DB".EDI."MODE BUFF" = 1) AND ("MODE SELECTION DB".EDI."PROCESS BUFF" = 2) AND ("EDI DB"."LEVEL HI RECIRC BUFF" = 3),
                     "PRESENT VALUE OF TIME" => "EDI DB"."RECIRCULATION ON TIMER PV");
END_REGION

REGION Network 15: AGAIN OFF TIME START AFTER RECIRCULATION OVER
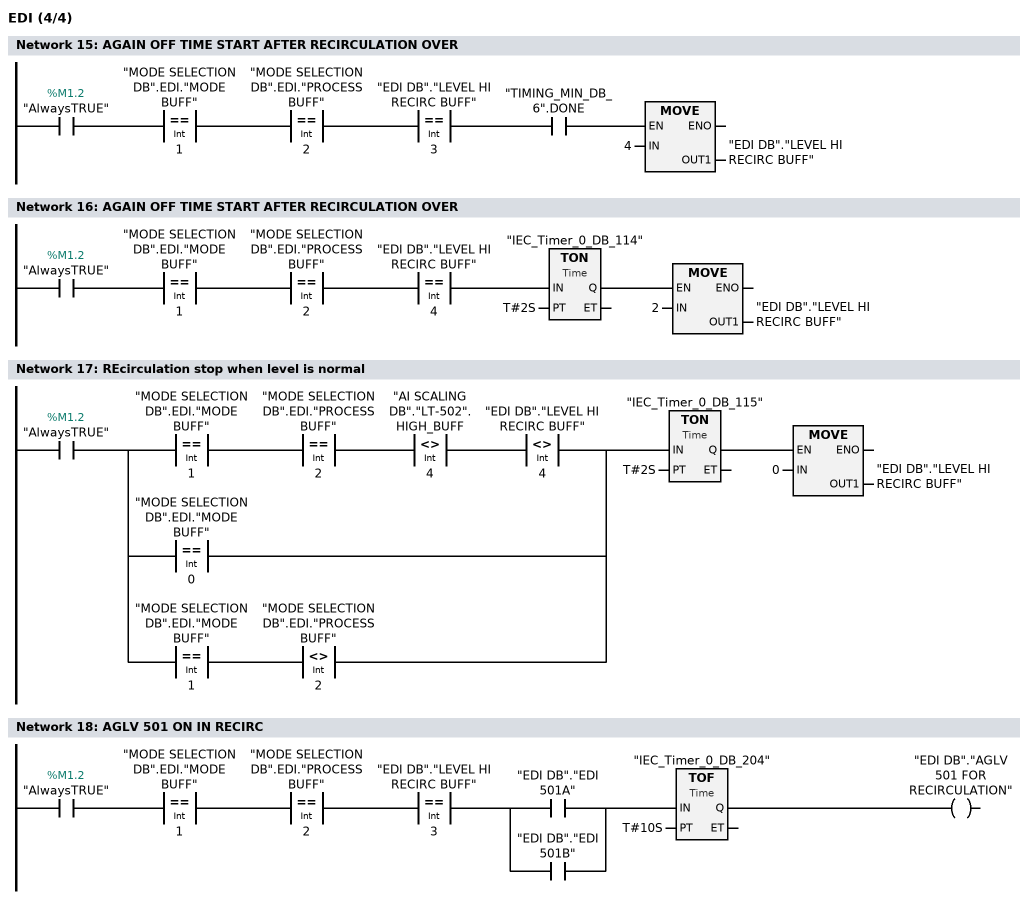
   RUNG wire#powerrail
      Contact( "AlwaysTRUE" )
      { S7_Templates := "SrcType := Int" } EQ_Contact(in1 := "MODE SELECTION DB".EDI."MODE BUFF", in2 := 1)
      { S7_Templates := "SrcType := Int" } EQ_Contact(in1 := "MODE SELECTION DB".EDI."PROCESS BUFF", in2 := 2)
      { S7_Templates := "SrcType := Int" } EQ_Contact(in1 := "EDI DB"."LEVEL HI RECIRC BUFF", in2 := 3)
      Contact( "TIMING_MIN_DB_6".DONE )
      Move(in := 4, out1 => "EDI DB"."LEVEL HI RECIRC BUFF")
   END_RUNG
   // the same network as SCL:
   IF "AlwaysTRUE" AND ("MODE SELECTION DB".EDI."MODE BUFF" = 1) AND ("MODE SELECTION DB".EDI."PROCESS BUFF" = 2) AND ("EDI DB"."LEVEL HI RECIRC BUFF" = 3) AND "TIMING_MIN_DB_6".DONE THEN
       "EDI DB"."LEVEL HI RECIRC BUFF" := 4;
   END_IF;
END_REGION

REGION Network 16: AGAIN OFF TIME START AFTER RECIRCULATION OVER
   RUNG wire#powerrail
      Contact( "AlwaysTRUE" )
      { S7_Templates := "SrcType := Int" } EQ_Contact(in1 := "MODE SELECTION DB".EDI."MODE BUFF", in2 := 1)
      { S7_Templates := "SrcType := Int" } EQ_Contact(in1 := "MODE SELECTION DB".EDI."PROCESS BUFF", in2 := 2)
      { S7_Templates := "SrcType := Int" } EQ_Contact(in1 := "EDI DB"."LEVEL HI RECIRC BUFF", in2 := 4)
      { S7_Templates := "time_type := Time" } "IEC_Timer_0_DB_114".TON(pt := T#2S, et =>)
      Move(in := 2, out1 => "EDI DB"."LEVEL HI RECIRC BUFF")
   END_RUNG
   // the same network as SCL:
   "IEC_Timer_0_DB_114".TON(IN := "AlwaysTRUE" AND ("MODE SELECTION DB".EDI."MODE BUFF" = 1) AND ("MODE SELECTION DB".EDI."PROCESS BUFF" = 2) AND ("EDI DB"."LEVEL HI RECIRC BUFF" = 4),
                           PT := T#2S);
   IF "IEC_Timer_0_DB_114".Q THEN "EDI DB"."LEVEL HI RECIRC BUFF" := 2; END_IF;
END_REGION

REGION Network 17: REcirculation stop when level is normal
   RUNG wire#powerrail
      Contact( "AlwaysTRUE" )
      wire#w1
      { S7_Templates := "SrcType := Int" } EQ_Contact(in1 := "MODE SELECTION DB".EDI."MODE BUFF", in2 := 1)
      { S7_Templates := "SrcType := Int" } EQ_Contact(in1 := "MODE SELECTION DB".EDI."PROCESS BUFF", in2 := 2)
      { S7_Templates := "SrcType := Int" } NE_Contact(in1 := "AI SCALING DB"."LT-502".HIGH_BUFF, in2 := 4)
      { S7_Templates := "SrcType := Int" } NE_Contact(in1 := "EDI DB"."LEVEL HI RECIRC BUFF", in2 := 4)
      wire#w2
      { S7_Templates := "time_type := Time" } "IEC_Timer_0_DB_115".TON(pt := T#2S, et =>)
      Move(in := 0, out1 => "EDI DB"."LEVEL HI RECIRC BUFF")
   END_RUNG
   RUNG wire#w1
      { S7_Templates := "SrcType := Int" } EQ_Contact(in1 := "MODE SELECTION DB".EDI."MODE BUFF", in2 := 0)
   END_RUNG wire#w2
   RUNG wire#w1
      { S7_Templates := "SrcType := Int" } EQ_Contact(in1 := "MODE SELECTION DB".EDI."MODE BUFF", in2 := 1)
      { S7_Templates := "SrcType := Int" } NE_Contact(in1 := "MODE SELECTION DB".EDI."PROCESS BUFF", in2 := 2)
   END_RUNG wire#w2
   // the same network as SCL:
   "IEC_Timer_0_DB_115".TON(IN := "AlwaysTRUE" AND ((("MODE SELECTION DB".EDI."MODE BUFF" = 1) AND ("MODE SELECTION DB".EDI."PROCESS BUFF" = 2) AND ("AI SCALING DB"."LT-502".HIGH_BUFF <> 4) AND ("EDI DB"."LEVEL HI RECIRC BUFF" <> 4)) OR ("MODE SELECTION DB".EDI."MODE BUFF" = 0) OR (("MODE SELECTION DB".EDI."MODE BUFF" = 1) AND ("MODE SELECTION DB".EDI."PROCESS BUFF" <> 2))),
                           PT := T#2S);
   IF "IEC_Timer_0_DB_115".Q THEN "EDI DB"."LEVEL HI RECIRC BUFF" := 0; END_IF;
END_REGION

REGION Network 18: AGLV 501 ON IN RECIRC
   RUNG wire#powerrail
      Contact( "AlwaysTRUE" )
      { S7_Templates := "SrcType := Int" } EQ_Contact(in1 := "MODE SELECTION DB".EDI."MODE BUFF", in2 := 1)
      { S7_Templates := "SrcType := Int" } EQ_Contact(in1 := "MODE SELECTION DB".EDI."PROCESS BUFF", in2 := 2)
      { S7_Templates := "SrcType := Int" } EQ_Contact(in1 := "EDI DB"."LEVEL HI RECIRC BUFF", in2 := 3)
      wire#w1
      Contact( "EDI DB"."EDI 501A" )
      wire#w2
      { S7_Templates := "time_type := Time" } "IEC_Timer_0_DB_204".TOF(pt := T#10S, et =>)
      Coil( "EDI DB"."AGLV 501 FOR RECIRCULATION" )
   END_RUNG
   RUNG wire#w1
      Contact( "EDI DB"."EDI 501B" )
   END_RUNG wire#w2
   // the same network as SCL:
   "IEC_Timer_0_DB_204".TOF(IN := "AlwaysTRUE" AND ("MODE SELECTION DB".EDI."MODE BUFF" = 1) AND ("MODE SELECTION DB".EDI."PROCESS BUFF" = 2) AND ("EDI DB"."LEVEL HI RECIRC BUFF" = 3) AND ("EDI DB"."EDI 501A" OR "EDI DB"."EDI 501B"),
                           PT := T#10S);
   "EDI DB"."AGLV 501 FOR RECIRCULATION" := "IEC_Timer_0_DB_204".Q;
END_REGION
END_FUNCTION

ORGANIZATION_BLOCK "MODBUS VFD"   // OB30, LAD, CyclicInterrupt
{ S7_Optimized_Access := 'TRUE' }
// stored: SetENOAutomatically false
   VAR_INPUT
      Initial_Call : Bool;   // Initial call of this OB
      Event_Count : Int;   // Events discarded
   END_VAR
   VAR_TEMP   // added for the SCL form of the ladder/FBD networks
      _w1 : Bool;
      _w2 : Bool;
   END_VAR
BEGIN

REGION Network 2: Slave 1 (SLAVE ID :- 1) WRITE
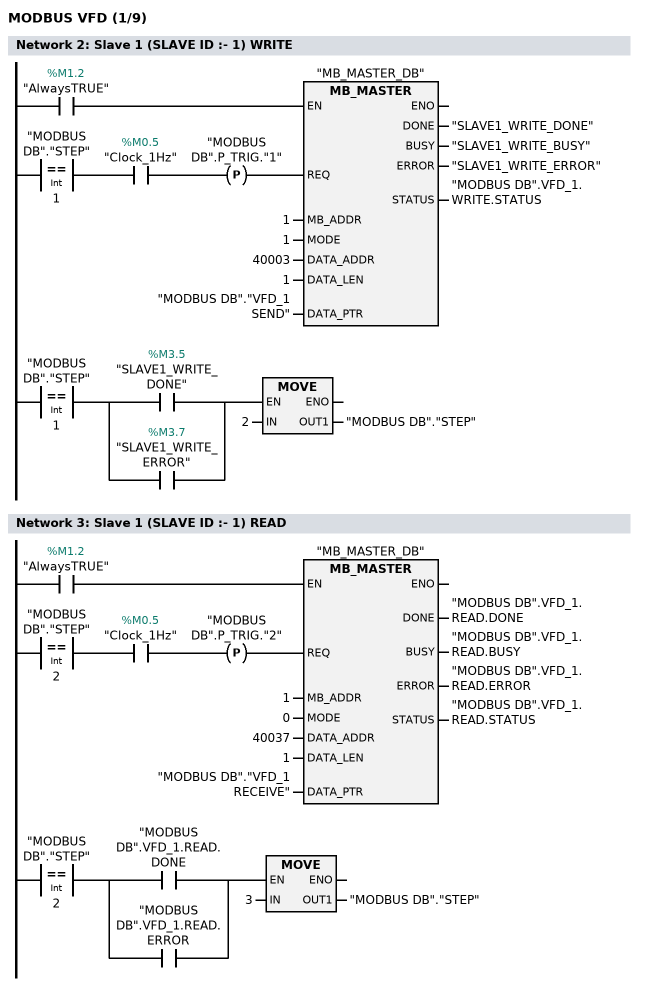
   RUNG wire#powerrail
      Contact( "AlwaysTRUE" )
      "MB_MASTER_DB".MB_MASTER(REQ := wire#w1, MB_ADDR := 1, MODE := 1, DATA_ADDR := 40003, DATA_LEN := 1, DATA_PTR := "MODBUS DB"."VFD_1 SEND", DONE => "SLAVE1_WRITE_DONE", BUSY => "SLAVE1_WRITE_BUSY", ERROR => "SLAVE1_WRITE_ERROR", STATUS => "MODBUS DB".VFD_1.WRITE.STATUS)
   END_RUNG
   RUNG wire#powerrail
      { S7_Templates := "SrcType := Int" } EQ_Contact(in1 := "MODBUS DB"."STEP", in2 := 1)
      Contact( "Clock_1Hz" )
      P_Trig( "MODBUS DB".P_TRIG."1" )
   END_RUNG wire#w1
   RUNG wire#powerrail
      { S7_Templates := "SrcType := Int" } EQ_Contact(in1 := "MODBUS DB"."STEP", in2 := 1)
      wire#w2
      Contact( "SLAVE1_WRITE_DONE" )
      wire#w3
      Move(in := 2, out1 => "MODBUS DB"."STEP")
   END_RUNG
   RUNG wire#w2
      Contact( "SLAVE1_WRITE_ERROR" )
   END_RUNG wire#w3
   // the same network as SCL:
   #_w1 := ("MODBUS DB"."STEP" = 1) AND "Clock_1Hz";
   #_w2 := #_w1 AND NOT "MODBUS DB".P_TRIG."1";   // rising edge
   "MODBUS DB".P_TRIG."1" := #_w1;
   IF "AlwaysTRUE" THEN
       "MB_MASTER_DB"(REQ := #_w2,   // MB_MASTER
                      MB_ADDR := 1,
                      MODE := 1,
                      DATA_ADDR := 40003,
                      DATA_LEN := 1,
                      DATA_PTR := "MODBUS DB"."VFD_1 SEND",
                      DONE => "SLAVE1_WRITE_DONE",
                      BUSY => "SLAVE1_WRITE_BUSY",
                      ERROR => "SLAVE1_WRITE_ERROR",
                      STATUS => "MODBUS DB".VFD_1.WRITE.STATUS);
   END_IF;
   IF ("MODBUS DB"."STEP" = 1) AND ("SLAVE1_WRITE_DONE" OR "SLAVE1_WRITE_ERROR") THEN
       "MODBUS DB"."STEP" := 2;
   END_IF;
END_REGION

REGION Network 3: Slave 1 (SLAVE ID :- 1) READ
   RUNG wire#powerrail
      Contact( "AlwaysTRUE" )
      "MB_MASTER_DB".MB_MASTER(REQ := wire#w1, MB_ADDR := 1, MODE := 0, DATA_ADDR := 40037, DATA_LEN := 1, DATA_PTR := "MODBUS DB"."VFD_1 RECEIVE", DONE => "MODBUS DB".VFD_1.READ.DONE, BUSY => "MODBUS DB".VFD_1.READ.BUSY, ERROR => "MODBUS DB".VFD_1.READ.ERROR, STATUS => "MODBUS DB".VFD_1.READ.STATUS)
   END_RUNG
   RUNG wire#powerrail
      { S7_Templates := "SrcType := Int" } EQ_Contact(in1 := "MODBUS DB"."STEP", in2 := 2)
      Contact( "Clock_1Hz" )
      P_Trig( "MODBUS DB".P_TRIG."2" )
   END_RUNG wire#w1
   RUNG wire#powerrail
      { S7_Templates := "SrcType := Int" } EQ_Contact(in1 := "MODBUS DB"."STEP", in2 := 2)
      wire#w2
      Contact( "MODBUS DB".VFD_1.READ.DONE )
      wire#w3
      Move(in := 3, out1 => "MODBUS DB"."STEP")
   END_RUNG
   RUNG wire#w2
      Contact( "MODBUS DB".VFD_1.READ.ERROR )
   END_RUNG wire#w3
   // the same network as SCL:
   #_w1 := ("MODBUS DB"."STEP" = 2) AND "Clock_1Hz";
   #_w2 := #_w1 AND NOT "MODBUS DB".P_TRIG."2";   // rising edge
   "MODBUS DB".P_TRIG."2" := #_w1;
   IF "AlwaysTRUE" THEN
       "MB_MASTER_DB"(REQ := #_w2,   // MB_MASTER
                      MB_ADDR := 1,
                      MODE := 0,
                      DATA_ADDR := 40037,
                      DATA_LEN := 1,
                      DATA_PTR := "MODBUS DB"."VFD_1 RECEIVE",
                      DONE => "MODBUS DB".VFD_1.READ.DONE,
                      BUSY => "MODBUS DB".VFD_1.READ.BUSY,
                      ERROR => "MODBUS DB".VFD_1.READ.ERROR,
                      STATUS => "MODBUS DB".VFD_1.READ.STATUS);
   END_IF;
   IF ("MODBUS DB"."STEP" = 2) AND ("MODBUS DB".VFD_1.READ.DONE OR "MODBUS DB".VFD_1.READ.ERROR) THEN
       "MODBUS DB"."STEP" := 3;
   END_IF;
END_REGION

REGION Network 4: Slave 2 (SLAVE ID :- 2) WRITE
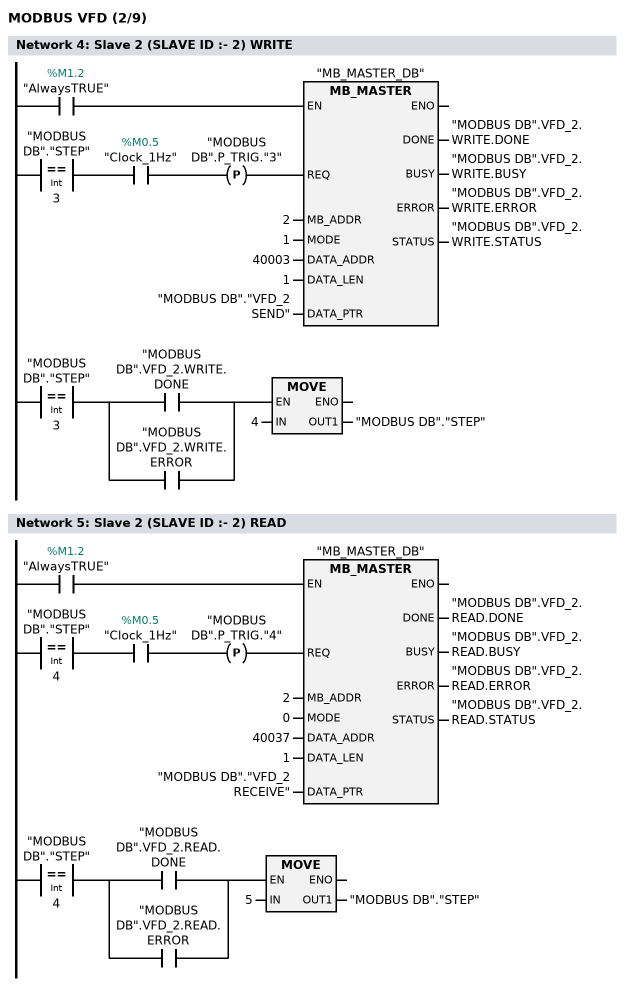
   RUNG wire#powerrail
      Contact( "AlwaysTRUE" )
      "MB_MASTER_DB".MB_MASTER(REQ := wire#w1, MB_ADDR := 2, MODE := 1, DATA_ADDR := 40003, DATA_LEN := 1, DATA_PTR := "MODBUS DB"."VFD_2 SEND", DONE => "MODBUS DB".VFD_2.WRITE.DONE, BUSY => "MODBUS DB".VFD_2.WRITE.BUSY, ERROR => "MODBUS DB".VFD_2.WRITE.ERROR, STATUS => "MODBUS DB".VFD_2.WRITE.STATUS)
   END_RUNG
   RUNG wire#powerrail
      { S7_Templates := "SrcType := Int" } EQ_Contact(in1 := "MODBUS DB"."STEP", in2 := 3)
      Contact( "Clock_1Hz" )
      P_Trig( "MODBUS DB".P_TRIG."3" )
   END_RUNG wire#w1
   RUNG wire#powerrail
      { S7_Templates := "SrcType := Int" } EQ_Contact(in1 := "MODBUS DB"."STEP", in2 := 3)
      wire#w2
      Contact( "MODBUS DB".VFD_2.WRITE.DONE )
      wire#w3
      Move(in := 4, out1 => "MODBUS DB"."STEP")
   END_RUNG
   RUNG wire#w2
      Contact( "MODBUS DB".VFD_2.WRITE.ERROR )
   END_RUNG wire#w3
   // the same network as SCL:
   #_w1 := ("MODBUS DB"."STEP" = 3) AND "Clock_1Hz";
   #_w2 := #_w1 AND NOT "MODBUS DB".P_TRIG."3";   // rising edge
   "MODBUS DB".P_TRIG."3" := #_w1;
   IF "AlwaysTRUE" THEN
       "MB_MASTER_DB"(REQ := #_w2,   // MB_MASTER
                      MB_ADDR := 2,
                      MODE := 1,
                      DATA_ADDR := 40003,
                      DATA_LEN := 1,
                      DATA_PTR := "MODBUS DB"."VFD_2 SEND",
                      DONE => "MODBUS DB".VFD_2.WRITE.DONE,
                      BUSY => "MODBUS DB".VFD_2.WRITE.BUSY,
                      ERROR => "MODBUS DB".VFD_2.WRITE.ERROR,
                      STATUS => "MODBUS DB".VFD_2.WRITE.STATUS);
   END_IF;
   IF ("MODBUS DB"."STEP" = 3) AND ("MODBUS DB".VFD_2.WRITE.DONE OR "MODBUS DB".VFD_2.WRITE.ERROR) THEN
       "MODBUS DB"."STEP" := 4;
   END_IF;
END_REGION

REGION Network 5: Slave 2 (SLAVE ID :- 2) READ
   RUNG wire#powerrail
      Contact( "AlwaysTRUE" )
      "MB_MASTER_DB".MB_MASTER(REQ := wire#w1, MB_ADDR := 2, MODE := 0, DATA_ADDR := 40037, DATA_LEN := 1, DATA_PTR := "MODBUS DB"."VFD_2 RECEIVE", DONE => "MODBUS DB".VFD_2.READ.DONE, BUSY => "MODBUS DB".VFD_2.READ.BUSY, ERROR => "MODBUS DB".VFD_2.READ.ERROR, STATUS => "MODBUS DB".VFD_2.READ.STATUS)
   END_RUNG
   RUNG wire#powerrail
      { S7_Templates := "SrcType := Int" } EQ_Contact(in1 := "MODBUS DB"."STEP", in2 := 4)
      Contact( "Clock_1Hz" )
      P_Trig( "MODBUS DB".P_TRIG."4" )
   END_RUNG wire#w1
   RUNG wire#powerrail
      { S7_Templates := "SrcType := Int" } EQ_Contact(in1 := "MODBUS DB"."STEP", in2 := 4)
      wire#w2
      Contact( "MODBUS DB".VFD_2.READ.DONE )
      wire#w3
      Move(in := 5, out1 => "MODBUS DB"."STEP")
   END_RUNG
   RUNG wire#w2
      Contact( "MODBUS DB".VFD_2.READ.ERROR )
   END_RUNG wire#w3
   // the same network as SCL:
   #_w1 := ("MODBUS DB"."STEP" = 4) AND "Clock_1Hz";
   #_w2 := #_w1 AND NOT "MODBUS DB".P_TRIG."4";   // rising edge
   "MODBUS DB".P_TRIG."4" := #_w1;
   IF "AlwaysTRUE" THEN
       "MB_MASTER_DB"(REQ := #_w2,   // MB_MASTER
                      MB_ADDR := 2,
                      MODE := 0,
                      DATA_ADDR := 40037,
                      DATA_LEN := 1,
                      DATA_PTR := "MODBUS DB"."VFD_2 RECEIVE",
                      DONE => "MODBUS DB".VFD_2.READ.DONE,
                      BUSY => "MODBUS DB".VFD_2.READ.BUSY,
                      ERROR => "MODBUS DB".VFD_2.READ.ERROR,
                      STATUS => "MODBUS DB".VFD_2.READ.STATUS);
   END_IF;
   IF ("MODBUS DB"."STEP" = 4) AND ("MODBUS DB".VFD_2.READ.DONE OR "MODBUS DB".VFD_2.READ.ERROR) THEN
       "MODBUS DB"."STEP" := 5;
   END_IF;
END_REGION

REGION Network 6: Slave 3 (SLAVE ID :- 3) WRITE
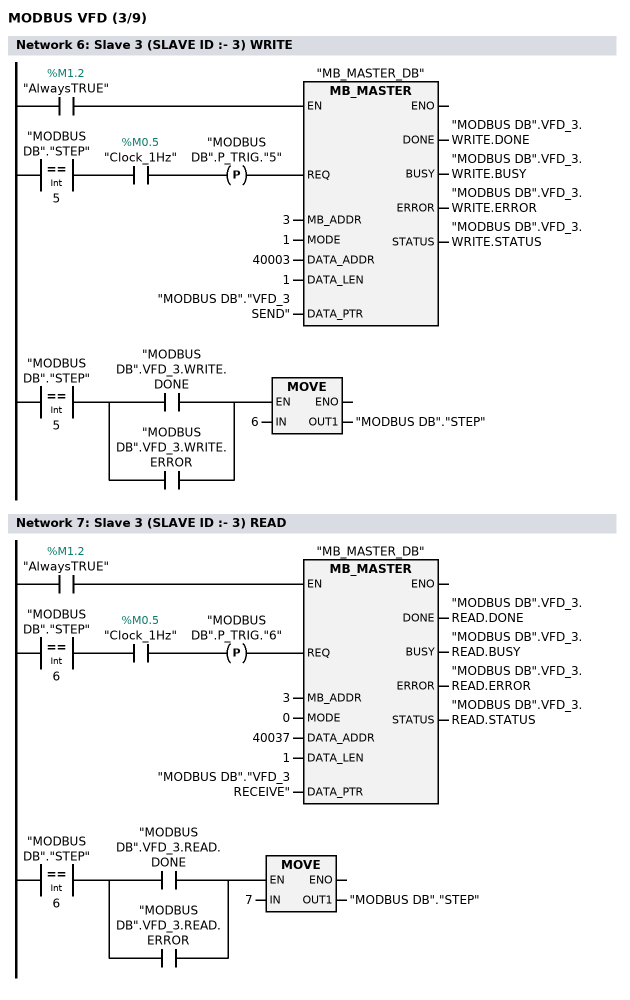
   RUNG wire#powerrail
      Contact( "AlwaysTRUE" )
      "MB_MASTER_DB".MB_MASTER(REQ := wire#w1, MB_ADDR := 3, MODE := 1, DATA_ADDR := 40003, DATA_LEN := 1, DATA_PTR := "MODBUS DB"."VFD_3 SEND", DONE => "MODBUS DB".VFD_3.WRITE.DONE, BUSY => "MODBUS DB".VFD_3.WRITE.BUSY, ERROR => "MODBUS DB".VFD_3.WRITE.ERROR, STATUS => "MODBUS DB".VFD_3.WRITE.STATUS)
   END_RUNG
   RUNG wire#powerrail
      { S7_Templates := "SrcType := Int" } EQ_Contact(in1 := "MODBUS DB"."STEP", in2 := 5)
      Contact( "Clock_1Hz" )
      P_Trig( "MODBUS DB".P_TRIG."5" )
   END_RUNG wire#w1
   RUNG wire#powerrail
      { S7_Templates := "SrcType := Int" } EQ_Contact(in1 := "MODBUS DB"."STEP", in2 := 5)
      wire#w2
      Contact( "MODBUS DB".VFD_3.WRITE.DONE )
      wire#w3
      Move(in := 6, out1 => "MODBUS DB"."STEP")
   END_RUNG
   RUNG wire#w2
      Contact( "MODBUS DB".VFD_3.WRITE.ERROR )
   END_RUNG wire#w3
   // the same network as SCL:
   #_w1 := ("MODBUS DB"."STEP" = 5) AND "Clock_1Hz";
   #_w2 := #_w1 AND NOT "MODBUS DB".P_TRIG."5";   // rising edge
   "MODBUS DB".P_TRIG."5" := #_w1;
   IF "AlwaysTRUE" THEN
       "MB_MASTER_DB"(REQ := #_w2,   // MB_MASTER
                      MB_ADDR := 3,
                      MODE := 1,
                      DATA_ADDR := 40003,
                      DATA_LEN := 1,
                      DATA_PTR := "MODBUS DB"."VFD_3 SEND",
                      DONE => "MODBUS DB".VFD_3.WRITE.DONE,
                      BUSY => "MODBUS DB".VFD_3.WRITE.BUSY,
                      ERROR => "MODBUS DB".VFD_3.WRITE.ERROR,
                      STATUS => "MODBUS DB".VFD_3.WRITE.STATUS);
   END_IF;
   IF ("MODBUS DB"."STEP" = 5) AND ("MODBUS DB".VFD_3.WRITE.DONE OR "MODBUS DB".VFD_3.WRITE.ERROR) THEN
       "MODBUS DB"."STEP" := 6;
   END_IF;
END_REGION

REGION Network 7: Slave 3 (SLAVE ID :- 3) READ
   RUNG wire#powerrail
      Contact( "AlwaysTRUE" )
      "MB_MASTER_DB".MB_MASTER(REQ := wire#w1, MB_ADDR := 3, MODE := 0, DATA_ADDR := 40037, DATA_LEN := 1, DATA_PTR := "MODBUS DB"."VFD_3 RECEIVE", DONE => "MODBUS DB".VFD_3.READ.DONE, BUSY => "MODBUS DB".VFD_3.READ.BUSY, ERROR => "MODBUS DB".VFD_3.READ.ERROR, STATUS => "MODBUS DB".VFD_3.READ.STATUS)
   END_RUNG
   RUNG wire#powerrail
      { S7_Templates := "SrcType := Int" } EQ_Contact(in1 := "MODBUS DB"."STEP", in2 := 6)
      Contact( "Clock_1Hz" )
      P_Trig( "MODBUS DB".P_TRIG."6" )
   END_RUNG wire#w1
   RUNG wire#powerrail
      { S7_Templates := "SrcType := Int" } EQ_Contact(in1 := "MODBUS DB"."STEP", in2 := 6)
      wire#w2
      Contact( "MODBUS DB".VFD_3.READ.DONE )
      wire#w3
      Move(in := 7, out1 => "MODBUS DB"."STEP")
   END_RUNG
   RUNG wire#w2
      Contact( "MODBUS DB".VFD_3.READ.ERROR )
   END_RUNG wire#w3
   // the same network as SCL:
   #_w1 := ("MODBUS DB"."STEP" = 6) AND "Clock_1Hz";
   #_w2 := #_w1 AND NOT "MODBUS DB".P_TRIG."6";   // rising edge
   "MODBUS DB".P_TRIG."6" := #_w1;
   IF "AlwaysTRUE" THEN
       "MB_MASTER_DB"(REQ := #_w2,   // MB_MASTER
                      MB_ADDR := 3,
                      MODE := 0,
                      DATA_ADDR := 40037,
                      DATA_LEN := 1,
                      DATA_PTR := "MODBUS DB"."VFD_3 RECEIVE",
                      DONE => "MODBUS DB".VFD_3.READ.DONE,
                      BUSY => "MODBUS DB".VFD_3.READ.BUSY,
                      ERROR => "MODBUS DB".VFD_3.READ.ERROR,
                      STATUS => "MODBUS DB".VFD_3.READ.STATUS);
   END_IF;
   IF ("MODBUS DB"."STEP" = 6) AND ("MODBUS DB".VFD_3.READ.DONE OR "MODBUS DB".VFD_3.READ.ERROR) THEN
       "MODBUS DB"."STEP" := 7;
   END_IF;
END_REGION

REGION Network 8: Slave 4 (SLAVE ID :- 4) WRITE
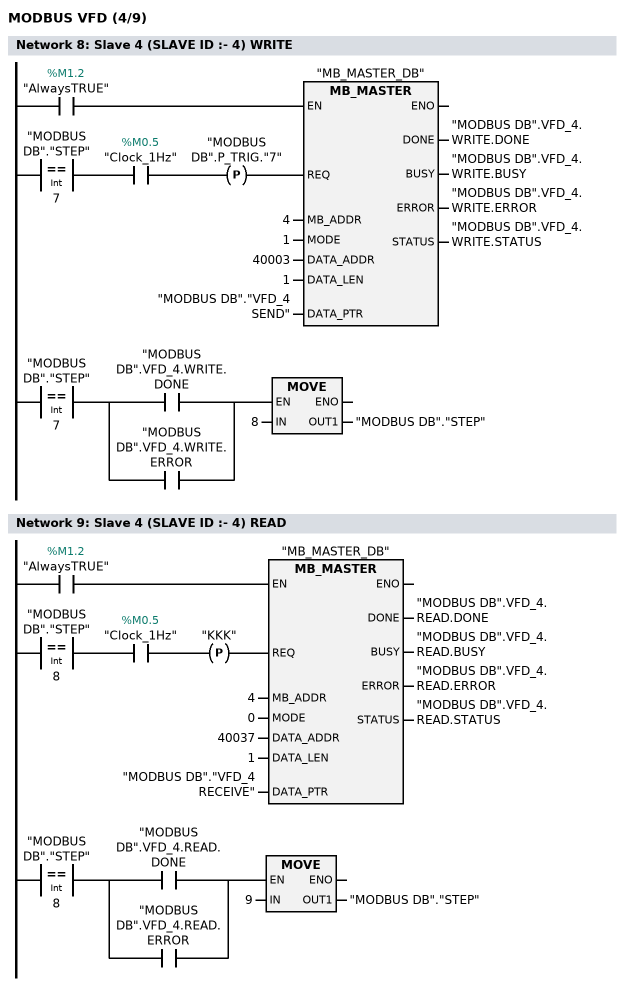
   RUNG wire#powerrail
      Contact( "AlwaysTRUE" )
      "MB_MASTER_DB".MB_MASTER(REQ := wire#w1, MB_ADDR := 4, MODE := 1, DATA_ADDR := 40003, DATA_LEN := 1, DATA_PTR := "MODBUS DB"."VFD_4 SEND", DONE => "MODBUS DB".VFD_4.WRITE.DONE, BUSY => "MODBUS DB".VFD_4.WRITE.BUSY, ERROR => "MODBUS DB".VFD_4.WRITE.ERROR, STATUS => "MODBUS DB".VFD_4.WRITE.STATUS)
   END_RUNG
   RUNG wire#powerrail
      { S7_Templates := "SrcType := Int" } EQ_Contact(in1 := "MODBUS DB"."STEP", in2 := 7)
      Contact( "Clock_1Hz" )
      P_Trig( "MODBUS DB".P_TRIG."7" )
   END_RUNG wire#w1
   RUNG wire#powerrail
      { S7_Templates := "SrcType := Int" } EQ_Contact(in1 := "MODBUS DB"."STEP", in2 := 7)
      wire#w2
      Contact( "MODBUS DB".VFD_4.WRITE.DONE )
      wire#w3
      Move(in := 8, out1 => "MODBUS DB"."STEP")
   END_RUNG
   RUNG wire#w2
      Contact( "MODBUS DB".VFD_4.WRITE.ERROR )
   END_RUNG wire#w3
   // the same network as SCL:
   #_w1 := ("MODBUS DB"."STEP" = 7) AND "Clock_1Hz";
   #_w2 := #_w1 AND NOT "MODBUS DB".P_TRIG."7";   // rising edge
   "MODBUS DB".P_TRIG."7" := #_w1;
   IF "AlwaysTRUE" THEN
       "MB_MASTER_DB"(REQ := #_w2,   // MB_MASTER
                      MB_ADDR := 4,
                      MODE := 1,
                      DATA_ADDR := 40003,
                      DATA_LEN := 1,
                      DATA_PTR := "MODBUS DB"."VFD_4 SEND",
                      DONE => "MODBUS DB".VFD_4.WRITE.DONE,
                      BUSY => "MODBUS DB".VFD_4.WRITE.BUSY,
                      ERROR => "MODBUS DB".VFD_4.WRITE.ERROR,
                      STATUS => "MODBUS DB".VFD_4.WRITE.STATUS);
   END_IF;
   IF ("MODBUS DB"."STEP" = 7) AND ("MODBUS DB".VFD_4.WRITE.DONE OR "MODBUS DB".VFD_4.WRITE.ERROR) THEN
       "MODBUS DB"."STEP" := 8;
   END_IF;
END_REGION

REGION Network 9: Slave 4 (SLAVE ID :- 4) READ
   RUNG wire#powerrail
      Contact( "AlwaysTRUE" )
      "MB_MASTER_DB".MB_MASTER(REQ := wire#w1, MB_ADDR := 4, MODE := 0, DATA_ADDR := 40037, DATA_LEN := 1, DATA_PTR := "MODBUS DB"."VFD_4 RECEIVE", DONE => "MODBUS DB".VFD_4.READ.DONE, BUSY => "MODBUS DB".VFD_4.READ.BUSY, ERROR => "MODBUS DB".VFD_4.READ.ERROR, STATUS => "MODBUS DB".VFD_4.READ.STATUS)
   END_RUNG
   RUNG wire#powerrail
      { S7_Templates := "SrcType := Int" } EQ_Contact(in1 := "MODBUS DB"."STEP", in2 := 8)
      Contact( "Clock_1Hz" )
      P_Trig( "KKK" )
   END_RUNG wire#w1
   RUNG wire#powerrail
      { S7_Templates := "SrcType := Int" } EQ_Contact(in1 := "MODBUS DB"."STEP", in2 := 8)
      wire#w2
      Contact( "MODBUS DB".VFD_4.READ.DONE )
      wire#w3
      Move(in := 9, out1 => "MODBUS DB"."STEP")
   END_RUNG
   RUNG wire#w2
      Contact( "MODBUS DB".VFD_4.READ.ERROR )
   END_RUNG wire#w3
   // the same network as SCL:
   #_w1 := ("MODBUS DB"."STEP" = 8) AND "Clock_1Hz";
   #_w2 := #_w1 AND NOT "KKK";   // rising edge
   "KKK" := #_w1;
   IF "AlwaysTRUE" THEN
       "MB_MASTER_DB"(REQ := #_w2,   // MB_MASTER
                      MB_ADDR := 4,
                      MODE := 0,
                      DATA_ADDR := 40037,
                      DATA_LEN := 1,
                      DATA_PTR := "MODBUS DB"."VFD_4 RECEIVE",
                      DONE => "MODBUS DB".VFD_4.READ.DONE,
                      BUSY => "MODBUS DB".VFD_4.READ.BUSY,
                      ERROR => "MODBUS DB".VFD_4.READ.ERROR,
                      STATUS => "MODBUS DB".VFD_4.READ.STATUS);
   END_IF;
   IF ("MODBUS DB"."STEP" = 8) AND ("MODBUS DB".VFD_4.READ.DONE OR "MODBUS DB".VFD_4.READ.ERROR) THEN
       "MODBUS DB"."STEP" := 9;
   END_IF;
END_REGION

REGION Network 10: Slave 5 (SLAVE ID :- 5) WRITE
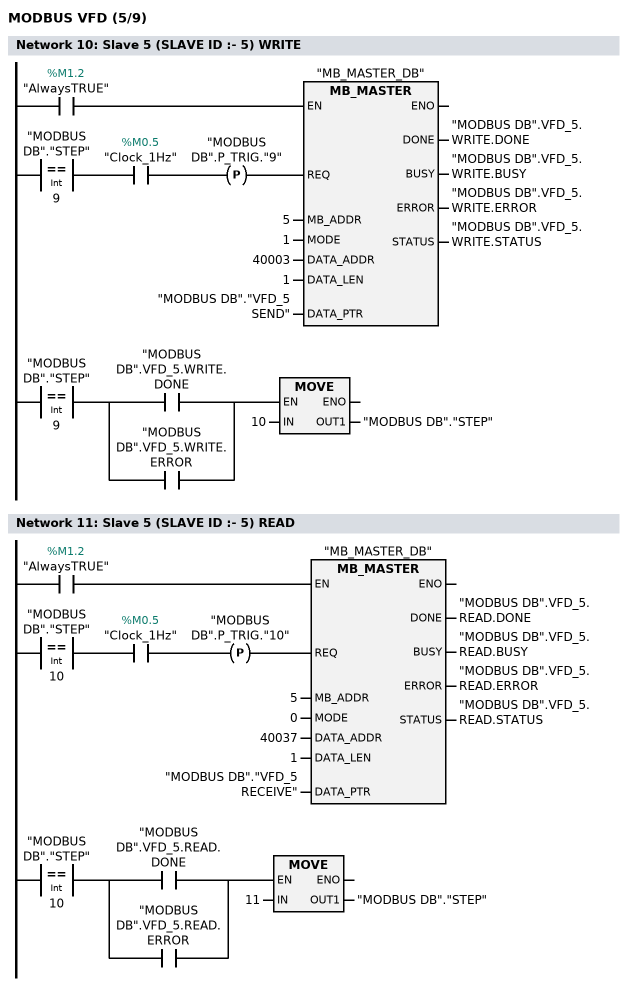
   RUNG wire#powerrail
      Contact( "AlwaysTRUE" )
      "MB_MASTER_DB".MB_MASTER(REQ := wire#w1, MB_ADDR := 5, MODE := 1, DATA_ADDR := 40003, DATA_LEN := 1, DATA_PTR := "MODBUS DB"."VFD_5 SEND", DONE => "MODBUS DB".VFD_5.WRITE.DONE, BUSY => "MODBUS DB".VFD_5.WRITE.BUSY, ERROR => "MODBUS DB".VFD_5.WRITE.ERROR, STATUS => "MODBUS DB".VFD_5.WRITE.STATUS)
   END_RUNG
   RUNG wire#powerrail
      { S7_Templates := "SrcType := Int" } EQ_Contact(in1 := "MODBUS DB"."STEP", in2 := 9)
      Contact( "Clock_1Hz" )
      P_Trig( "MODBUS DB".P_TRIG."9" )
   END_RUNG wire#w1
   RUNG wire#powerrail
      { S7_Templates := "SrcType := Int" } EQ_Contact(in1 := "MODBUS DB"."STEP", in2 := 9)
      wire#w2
      Contact( "MODBUS DB".VFD_5.WRITE.DONE )
      wire#w3
      Move(in := 10, out1 => "MODBUS DB"."STEP")
   END_RUNG
   RUNG wire#w2
      Contact( "MODBUS DB".VFD_5.WRITE.ERROR )
   END_RUNG wire#w3
   // the same network as SCL:
   #_w1 := ("MODBUS DB"."STEP" = 9) AND "Clock_1Hz";
   #_w2 := #_w1 AND NOT "MODBUS DB".P_TRIG."9";   // rising edge
   "MODBUS DB".P_TRIG."9" := #_w1;
   IF "AlwaysTRUE" THEN
       "MB_MASTER_DB"(REQ := #_w2,   // MB_MASTER
                      MB_ADDR := 5,
                      MODE := 1,
                      DATA_ADDR := 40003,
                      DATA_LEN := 1,
                      DATA_PTR := "MODBUS DB"."VFD_5 SEND",
                      DONE => "MODBUS DB".VFD_5.WRITE.DONE,
                      BUSY => "MODBUS DB".VFD_5.WRITE.BUSY,
                      ERROR => "MODBUS DB".VFD_5.WRITE.ERROR,
                      STATUS => "MODBUS DB".VFD_5.WRITE.STATUS);
   END_IF;
   IF ("MODBUS DB"."STEP" = 9) AND ("MODBUS DB".VFD_5.WRITE.DONE OR "MODBUS DB".VFD_5.WRITE.ERROR) THEN
       "MODBUS DB"."STEP" := 10;
   END_IF;
END_REGION

REGION Network 11: Slave 5 (SLAVE ID :- 5) READ
   RUNG wire#powerrail
      Contact( "AlwaysTRUE" )
      "MB_MASTER_DB".MB_MASTER(REQ := wire#w1, MB_ADDR := 5, MODE := 0, DATA_ADDR := 40037, DATA_LEN := 1, DATA_PTR := "MODBUS DB"."VFD_5 RECEIVE", DONE => "MODBUS DB".VFD_5.READ.DONE, BUSY => "MODBUS DB".VFD_5.READ.BUSY, ERROR => "MODBUS DB".VFD_5.READ.ERROR, STATUS => "MODBUS DB".VFD_5.READ.STATUS)
   END_RUNG
   RUNG wire#powerrail
      { S7_Templates := "SrcType := Int" } EQ_Contact(in1 := "MODBUS DB"."STEP", in2 := 10)
      Contact( "Clock_1Hz" )
      P_Trig( "MODBUS DB".P_TRIG."10" )
   END_RUNG wire#w1
   RUNG wire#powerrail
      { S7_Templates := "SrcType := Int" } EQ_Contact(in1 := "MODBUS DB"."STEP", in2 := 10)
      wire#w2
      Contact( "MODBUS DB".VFD_5.READ.DONE )
      wire#w3
      Move(in := 11, out1 => "MODBUS DB"."STEP")
   END_RUNG
   RUNG wire#w2
      Contact( "MODBUS DB".VFD_5.READ.ERROR )
   END_RUNG wire#w3
   // the same network as SCL:
   #_w1 := ("MODBUS DB"."STEP" = 10) AND "Clock_1Hz";
   #_w2 := #_w1 AND NOT "MODBUS DB".P_TRIG."10";   // rising edge
   "MODBUS DB".P_TRIG."10" := #_w1;
   IF "AlwaysTRUE" THEN
       "MB_MASTER_DB"(REQ := #_w2,   // MB_MASTER
                      MB_ADDR := 5,
                      MODE := 0,
                      DATA_ADDR := 40037,
                      DATA_LEN := 1,
                      DATA_PTR := "MODBUS DB"."VFD_5 RECEIVE",
                      DONE => "MODBUS DB".VFD_5.READ.DONE,
                      BUSY => "MODBUS DB".VFD_5.READ.BUSY,
                      ERROR => "MODBUS DB".VFD_5.READ.ERROR,
                      STATUS => "MODBUS DB".VFD_5.READ.STATUS);
   END_IF;
   IF ("MODBUS DB"."STEP" = 10) AND ("MODBUS DB".VFD_5.READ.DONE OR "MODBUS DB".VFD_5.READ.ERROR) THEN
       "MODBUS DB"."STEP" := 11;
   END_IF;
END_REGION

REGION Network 12: Slave 6 (SLAVE ID :- 6) WRITE
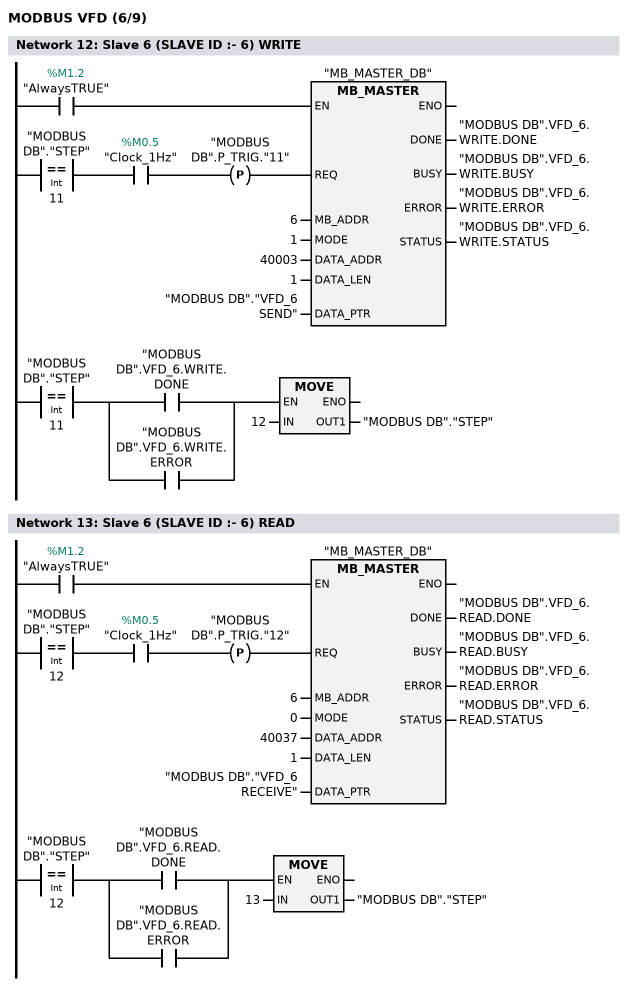
   RUNG wire#powerrail
      Contact( "AlwaysTRUE" )
      "MB_MASTER_DB".MB_MASTER(REQ := wire#w1, MB_ADDR := 6, MODE := 1, DATA_ADDR := 40003, DATA_LEN := 1, DATA_PTR := "MODBUS DB"."VFD_6 SEND", DONE => "MODBUS DB".VFD_6.WRITE.DONE, BUSY => "MODBUS DB".VFD_6.WRITE.BUSY, ERROR => "MODBUS DB".VFD_6.WRITE.ERROR, STATUS => "MODBUS DB".VFD_6.WRITE.STATUS)
   END_RUNG
   RUNG wire#powerrail
      { S7_Templates := "SrcType := Int" } EQ_Contact(in1 := "MODBUS DB"."STEP", in2 := 11)
      Contact( "Clock_1Hz" )
      P_Trig( "MODBUS DB".P_TRIG."11" )
   END_RUNG wire#w1
   RUNG wire#powerrail
      { S7_Templates := "SrcType := Int" } EQ_Contact(in1 := "MODBUS DB"."STEP", in2 := 11)
      wire#w2
      Contact( "MODBUS DB".VFD_6.WRITE.DONE )
      wire#w3
      Move(in := 12, out1 => "MODBUS DB"."STEP")
   END_RUNG
   RUNG wire#w2
      Contact( "MODBUS DB".VFD_6.WRITE.ERROR )
   END_RUNG wire#w3
   // the same network as SCL:
   #_w1 := ("MODBUS DB"."STEP" = 11) AND "Clock_1Hz";
   #_w2 := #_w1 AND NOT "MODBUS DB".P_TRIG."11";   // rising edge
   "MODBUS DB".P_TRIG."11" := #_w1;
   IF "AlwaysTRUE" THEN
       "MB_MASTER_DB"(REQ := #_w2,   // MB_MASTER
                      MB_ADDR := 6,
                      MODE := 1,
                      DATA_ADDR := 40003,
                      DATA_LEN := 1,
                      DATA_PTR := "MODBUS DB"."VFD_6 SEND",
                      DONE => "MODBUS DB".VFD_6.WRITE.DONE,
                      BUSY => "MODBUS DB".VFD_6.WRITE.BUSY,
                      ERROR => "MODBUS DB".VFD_6.WRITE.ERROR,
                      STATUS => "MODBUS DB".VFD_6.WRITE.STATUS);
   END_IF;
   IF ("MODBUS DB"."STEP" = 11) AND ("MODBUS DB".VFD_6.WRITE.DONE OR "MODBUS DB".VFD_6.WRITE.ERROR) THEN
       "MODBUS DB"."STEP" := 12;
   END_IF;
END_REGION

REGION Network 13: Slave 6 (SLAVE ID :- 6) READ
   RUNG wire#powerrail
      Contact( "AlwaysTRUE" )
      "MB_MASTER_DB".MB_MASTER(REQ := wire#w1, MB_ADDR := 6, MODE := 0, DATA_ADDR := 40037, DATA_LEN := 1, DATA_PTR := "MODBUS DB"."VFD_6 RECEIVE", DONE => "MODBUS DB".VFD_6.READ.DONE, BUSY => "MODBUS DB".VFD_6.READ.BUSY, ERROR => "MODBUS DB".VFD_6.READ.ERROR, STATUS => "MODBUS DB".VFD_6.READ.STATUS)
   END_RUNG
   RUNG wire#powerrail
      { S7_Templates := "SrcType := Int" } EQ_Contact(in1 := "MODBUS DB"."STEP", in2 := 12)
      Contact( "Clock_1Hz" )
      P_Trig( "MODBUS DB".P_TRIG."12" )
   END_RUNG wire#w1
   RUNG wire#powerrail
      { S7_Templates := "SrcType := Int" } EQ_Contact(in1 := "MODBUS DB"."STEP", in2 := 12)
      wire#w2
      Contact( "MODBUS DB".VFD_6.READ.DONE )
      wire#w3
      Move(in := 13, out1 => "MODBUS DB"."STEP")
   END_RUNG
   RUNG wire#w2
      Contact( "MODBUS DB".VFD_6.READ.ERROR )
   END_RUNG wire#w3
   // the same network as SCL:
   #_w1 := ("MODBUS DB"."STEP" = 12) AND "Clock_1Hz";
   #_w2 := #_w1 AND NOT "MODBUS DB".P_TRIG."12";   // rising edge
   "MODBUS DB".P_TRIG."12" := #_w1;
   IF "AlwaysTRUE" THEN
       "MB_MASTER_DB"(REQ := #_w2,   // MB_MASTER
                      MB_ADDR := 6,
                      MODE := 0,
                      DATA_ADDR := 40037,
                      DATA_LEN := 1,
                      DATA_PTR := "MODBUS DB"."VFD_6 RECEIVE",
                      DONE => "MODBUS DB".VFD_6.READ.DONE,
                      BUSY => "MODBUS DB".VFD_6.READ.BUSY,
                      ERROR => "MODBUS DB".VFD_6.READ.ERROR,
                      STATUS => "MODBUS DB".VFD_6.READ.STATUS);
   END_IF;
   IF ("MODBUS DB"."STEP" = 12) AND ("MODBUS DB".VFD_6.READ.DONE OR "MODBUS DB".VFD_6.READ.ERROR) THEN
       "MODBUS DB"."STEP" := 13;
   END_IF;
END_REGION

REGION Network 14: Slave 7 (SLAVE ID :- 7) WRITE
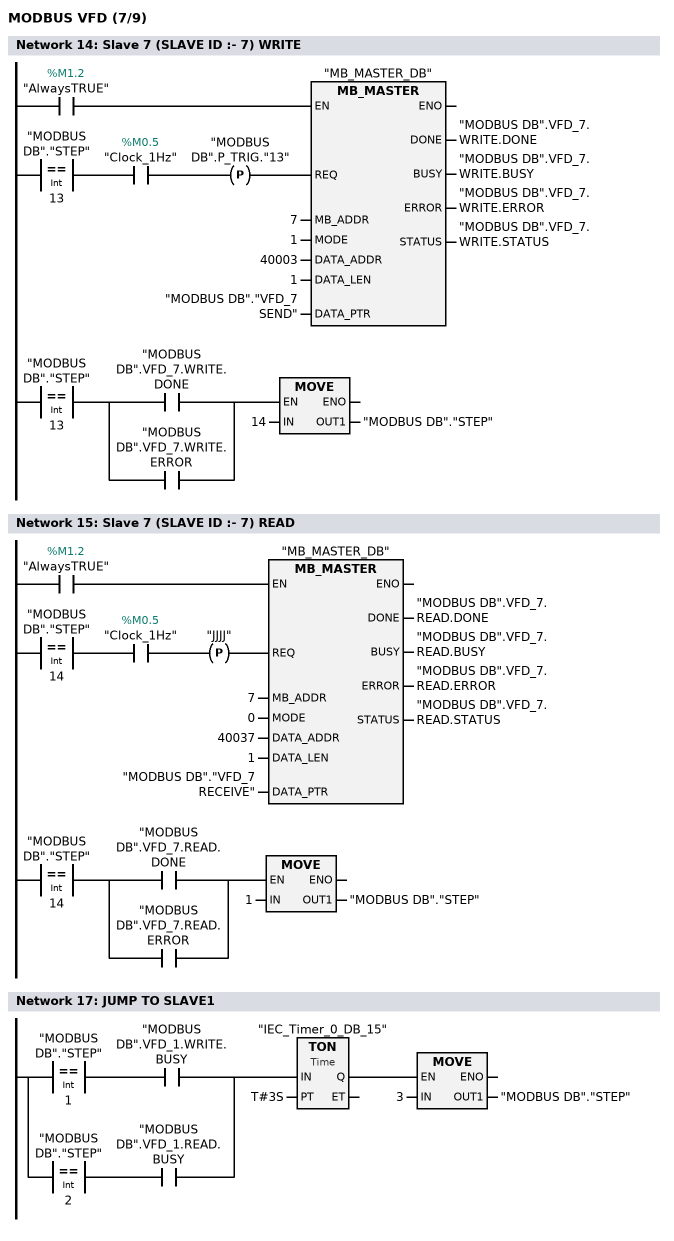
   RUNG wire#powerrail
      Contact( "AlwaysTRUE" )
      "MB_MASTER_DB".MB_MASTER(REQ := wire#w1, MB_ADDR := 7, MODE := 1, DATA_ADDR := 40003, DATA_LEN := 1, DATA_PTR := "MODBUS DB"."VFD_7 SEND", DONE => "MODBUS DB".VFD_7.WRITE.DONE, BUSY => "MODBUS DB".VFD_7.WRITE.BUSY, ERROR => "MODBUS DB".VFD_7.WRITE.ERROR, STATUS => "MODBUS DB".VFD_7.WRITE.STATUS)
   END_RUNG
   RUNG wire#powerrail
      { S7_Templates := "SrcType := Int" } EQ_Contact(in1 := "MODBUS DB"."STEP", in2 := 13)
      Contact( "Clock_1Hz" )
      P_Trig( "MODBUS DB".P_TRIG."13" )
   END_RUNG wire#w1
   RUNG wire#powerrail
      { S7_Templates := "SrcType := Int" } EQ_Contact(in1 := "MODBUS DB"."STEP", in2 := 13)
      wire#w2
      Contact( "MODBUS DB".VFD_7.WRITE.DONE )
      wire#w3
      Move(in := 14, out1 => "MODBUS DB"."STEP")
   END_RUNG
   RUNG wire#w2
      Contact( "MODBUS DB".VFD_7.WRITE.ERROR )
   END_RUNG wire#w3
   // the same network as SCL:
   #_w1 := ("MODBUS DB"."STEP" = 13) AND "Clock_1Hz";
   #_w2 := #_w1 AND NOT "MODBUS DB".P_TRIG."13";   // rising edge
   "MODBUS DB".P_TRIG."13" := #_w1;
   IF "AlwaysTRUE" THEN
       "MB_MASTER_DB"(REQ := #_w2,   // MB_MASTER
                      MB_ADDR := 7,
                      MODE := 1,
                      DATA_ADDR := 40003,
                      DATA_LEN := 1,
                      DATA_PTR := "MODBUS DB"."VFD_7 SEND",
                      DONE => "MODBUS DB".VFD_7.WRITE.DONE,
                      BUSY => "MODBUS DB".VFD_7.WRITE.BUSY,
                      ERROR => "MODBUS DB".VFD_7.WRITE.ERROR,
                      STATUS => "MODBUS DB".VFD_7.WRITE.STATUS);
   END_IF;
   IF ("MODBUS DB"."STEP" = 13) AND ("MODBUS DB".VFD_7.WRITE.DONE OR "MODBUS DB".VFD_7.WRITE.ERROR) THEN
       "MODBUS DB"."STEP" := 14;
   END_IF;
END_REGION

REGION Network 15: Slave 7 (SLAVE ID :- 7) READ
   RUNG wire#powerrail
      Contact( "AlwaysTRUE" )
      "MB_MASTER_DB".MB_MASTER(REQ := wire#w1, MB_ADDR := 7, MODE := 0, DATA_ADDR := 40037, DATA_LEN := 1, DATA_PTR := "MODBUS DB"."VFD_7 RECEIVE", DONE => "MODBUS DB".VFD_7.READ.DONE, BUSY => "MODBUS DB".VFD_7.READ.BUSY, ERROR => "MODBUS DB".VFD_7.READ.ERROR, STATUS => "MODBUS DB".VFD_7.READ.STATUS)
   END_RUNG
   RUNG wire#powerrail
      { S7_Templates := "SrcType := Int" } EQ_Contact(in1 := "MODBUS DB"."STEP", in2 := 14)
      Contact( "Clock_1Hz" )
      P_Trig( "JJJJ" )
   END_RUNG wire#w1
   RUNG wire#powerrail
      { S7_Templates := "SrcType := Int" } EQ_Contact(in1 := "MODBUS DB"."STEP", in2 := 14)
      wire#w2
      Contact( "MODBUS DB".VFD_7.READ.DONE )
      wire#w3
      Move(in := 1, out1 => "MODBUS DB"."STEP")
   END_RUNG
   RUNG wire#w2
      Contact( "MODBUS DB".VFD_7.READ.ERROR )
   END_RUNG wire#w3
   // the same network as SCL:
   #_w1 := ("MODBUS DB"."STEP" = 14) AND "Clock_1Hz";
   #_w2 := #_w1 AND NOT "JJJJ";   // rising edge
   "JJJJ" := #_w1;
   IF "AlwaysTRUE" THEN
       "MB_MASTER_DB"(REQ := #_w2,   // MB_MASTER
                      MB_ADDR := 7,
                      MODE := 0,
                      DATA_ADDR := 40037,
                      DATA_LEN := 1,
                      DATA_PTR := "MODBUS DB"."VFD_7 RECEIVE",
                      DONE => "MODBUS DB".VFD_7.READ.DONE,
                      BUSY => "MODBUS DB".VFD_7.READ.BUSY,
                      ERROR => "MODBUS DB".VFD_7.READ.ERROR,
                      STATUS => "MODBUS DB".VFD_7.READ.STATUS);
   END_IF;
   IF ("MODBUS DB"."STEP" = 14) AND ("MODBUS DB".VFD_7.READ.DONE OR "MODBUS DB".VFD_7.READ.ERROR) THEN
       "MODBUS DB"."STEP" := 1;
   END_IF;
END_REGION

REGION Network 17: JUMP TO SLAVE1
   RUNG wire#powerrail
      { S7_Templates := "SrcType := Int" } EQ_Contact(in1 := "MODBUS DB"."STEP", in2 := 1)
      Contact( "MODBUS DB".VFD_1.WRITE.BUSY )
      wire#w1
      { S7_Templates := "time_type := Time" } "IEC_Timer_0_DB_15".TON(pt := T#3S, et =>)
      Move(in := 3, out1 => "MODBUS DB"."STEP")
   END_RUNG
   RUNG wire#powerrail
      { S7_Templates := "SrcType := Int" } EQ_Contact(in1 := "MODBUS DB"."STEP", in2 := 2)
      Contact( "MODBUS DB".VFD_1.READ.BUSY )
   END_RUNG wire#w1
   // the same network as SCL:
   "IEC_Timer_0_DB_15".TON(IN := (("MODBUS DB"."STEP" = 1) AND "MODBUS DB".VFD_1.WRITE.BUSY) OR (("MODBUS DB"."STEP" = 2) AND "MODBUS DB".VFD_1.READ.BUSY),
                           PT := T#3S);
   IF "IEC_Timer_0_DB_15".Q THEN "MODBUS DB"."STEP" := 3; END_IF;
END_REGION

REGION Network 18: JUMP TO SLAVE2
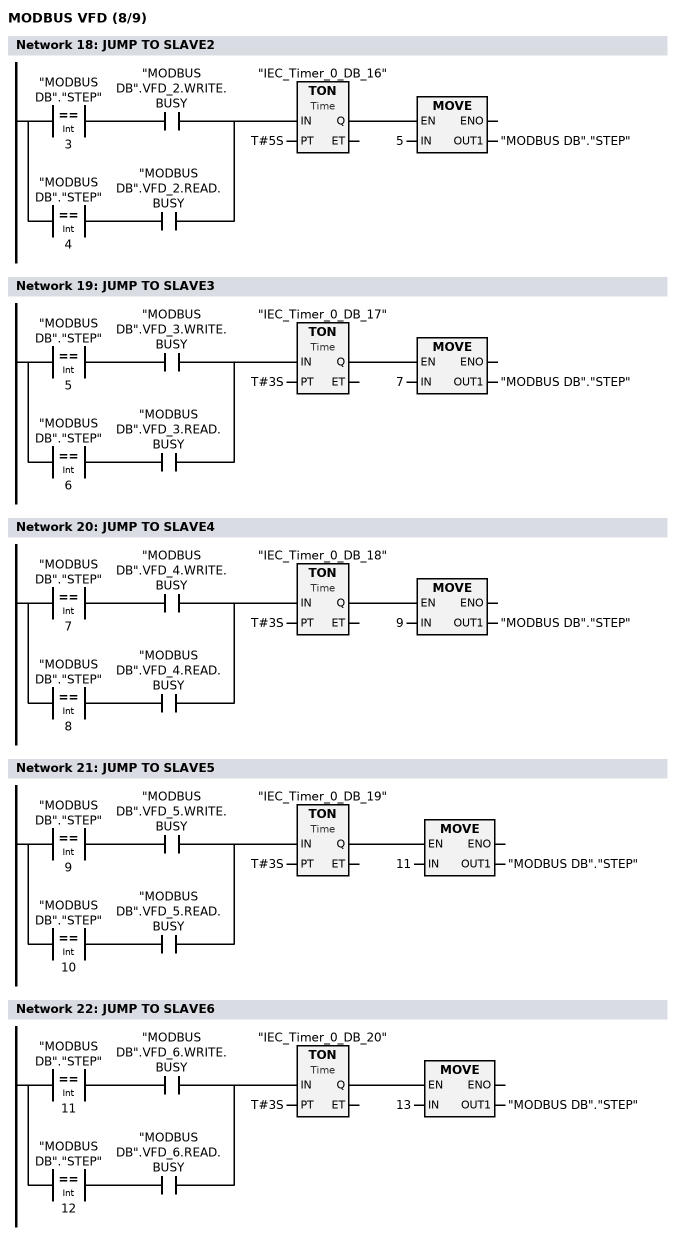
   RUNG wire#powerrail
      { S7_Templates := "SrcType := Int" } EQ_Contact(in1 := "MODBUS DB"."STEP", in2 := 3)
      Contact( "MODBUS DB".VFD_2.WRITE.BUSY )
      wire#w1
      { S7_Templates := "time_type := Time" } "IEC_Timer_0_DB_16".TON(pt := T#5S, et =>)
      Move(in := 5, out1 => "MODBUS DB"."STEP")
   END_RUNG
   RUNG wire#powerrail
      { S7_Templates := "SrcType := Int" } EQ_Contact(in1 := "MODBUS DB"."STEP", in2 := 4)
      Contact( "MODBUS DB".VFD_2.READ.BUSY )
   END_RUNG wire#w1
   // the same network as SCL:
   "IEC_Timer_0_DB_16".TON(IN := (("MODBUS DB"."STEP" = 3) AND "MODBUS DB".VFD_2.WRITE.BUSY) OR (("MODBUS DB"."STEP" = 4) AND "MODBUS DB".VFD_2.READ.BUSY),
                           PT := T#5S);
   IF "IEC_Timer_0_DB_16".Q THEN "MODBUS DB"."STEP" := 5; END_IF;
END_REGION

REGION Network 19: JUMP TO SLAVE3
   RUNG wire#powerrail
      { S7_Templates := "SrcType := Int" } EQ_Contact(in1 := "MODBUS DB"."STEP", in2 := 5)
      Contact( "MODBUS DB".VFD_3.WRITE.BUSY )
      wire#w1
      { S7_Templates := "time_type := Time" } "IEC_Timer_0_DB_17".TON(pt := T#3S, et =>)
      Move(in := 7, out1 => "MODBUS DB"."STEP")
   END_RUNG
   RUNG wire#powerrail
      { S7_Templates := "SrcType := Int" } EQ_Contact(in1 := "MODBUS DB"."STEP", in2 := 6)
      Contact( "MODBUS DB".VFD_3.READ.BUSY )
   END_RUNG wire#w1
   // the same network as SCL:
   "IEC_Timer_0_DB_17".TON(IN := (("MODBUS DB"."STEP" = 5) AND "MODBUS DB".VFD_3.WRITE.BUSY) OR (("MODBUS DB"."STEP" = 6) AND "MODBUS DB".VFD_3.READ.BUSY),
                           PT := T#3S);
   IF "IEC_Timer_0_DB_17".Q THEN "MODBUS DB"."STEP" := 7; END_IF;
END_REGION

REGION Network 20: JUMP TO SLAVE4
   RUNG wire#powerrail
      { S7_Templates := "SrcType := Int" } EQ_Contact(in1 := "MODBUS DB"."STEP", in2 := 7)
      Contact( "MODBUS DB".VFD_4.WRITE.BUSY )
      wire#w1
      { S7_Templates := "time_type := Time" } "IEC_Timer_0_DB_18".TON(pt := T#3S, et =>)
      Move(in := 9, out1 => "MODBUS DB"."STEP")
   END_RUNG
   RUNG wire#powerrail
      { S7_Templates := "SrcType := Int" } EQ_Contact(in1 := "MODBUS DB"."STEP", in2 := 8)
      Contact( "MODBUS DB".VFD_4.READ.BUSY )
   END_RUNG wire#w1
   // the same network as SCL:
   "IEC_Timer_0_DB_18".TON(IN := (("MODBUS DB"."STEP" = 7) AND "MODBUS DB".VFD_4.WRITE.BUSY) OR (("MODBUS DB"."STEP" = 8) AND "MODBUS DB".VFD_4.READ.BUSY),
                           PT := T#3S);
   IF "IEC_Timer_0_DB_18".Q THEN "MODBUS DB"."STEP" := 9; END_IF;
END_REGION

REGION Network 21: JUMP TO SLAVE5
   RUNG wire#powerrail
      { S7_Templates := "SrcType := Int" } EQ_Contact(in1 := "MODBUS DB"."STEP", in2 := 9)
      Contact( "MODBUS DB".VFD_5.WRITE.BUSY )
      wire#w1
      { S7_Templates := "time_type := Time" } "IEC_Timer_0_DB_19".TON(pt := T#3S, et =>)
      Move(in := 11, out1 => "MODBUS DB"."STEP")
   END_RUNG
   RUNG wire#powerrail
      { S7_Templates := "SrcType := Int" } EQ_Contact(in1 := "MODBUS DB"."STEP", in2 := 10)
      Contact( "MODBUS DB".VFD_5.READ.BUSY )
   END_RUNG wire#w1
   // the same network as SCL:
   "IEC_Timer_0_DB_19".TON(IN := (("MODBUS DB"."STEP" = 9) AND "MODBUS DB".VFD_5.WRITE.BUSY) OR (("MODBUS DB"."STEP" = 10) AND "MODBUS DB".VFD_5.READ.BUSY),
                           PT := T#3S);
   IF "IEC_Timer_0_DB_19".Q THEN "MODBUS DB"."STEP" := 11; END_IF;
END_REGION

REGION Network 22: JUMP TO SLAVE6
   RUNG wire#powerrail
      { S7_Templates := "SrcType := Int" } EQ_Contact(in1 := "MODBUS DB"."STEP", in2 := 11)
      Contact( "MODBUS DB".VFD_6.WRITE.BUSY )
      wire#w1
      { S7_Templates := "time_type := Time" } "IEC_Timer_0_DB_20".TON(pt := T#3S, et =>)
      Move(in := 13, out1 => "MODBUS DB"."STEP")
   END_RUNG
   RUNG wire#powerrail
      { S7_Templates := "SrcType := Int" } EQ_Contact(in1 := "MODBUS DB"."STEP", in2 := 12)
      Contact( "MODBUS DB".VFD_6.READ.BUSY )
   END_RUNG wire#w1
   // the same network as SCL:
   "IEC_Timer_0_DB_20".TON(IN := (("MODBUS DB"."STEP" = 11) AND "MODBUS DB".VFD_6.WRITE.BUSY) OR (("MODBUS DB"."STEP" = 12) AND "MODBUS DB".VFD_6.READ.BUSY),
                           PT := T#3S);
   IF "IEC_Timer_0_DB_20".Q THEN "MODBUS DB"."STEP" := 13; END_IF;
END_REGION

REGION Network 23: JUMP TO SLAVE7
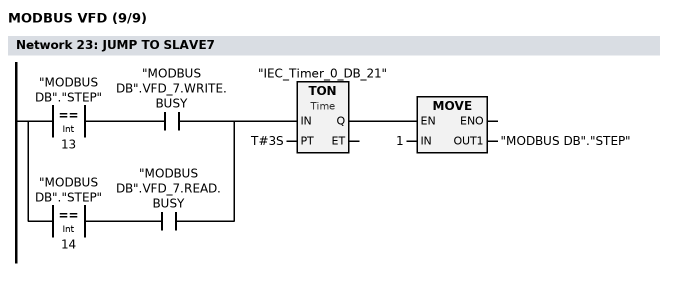
   RUNG wire#powerrail
      { S7_Templates := "SrcType := Int" } EQ_Contact(in1 := "MODBUS DB"."STEP", in2 := 13)
      Contact( "MODBUS DB".VFD_7.WRITE.BUSY )
      wire#w1
      { S7_Templates := "time_type := Time" } "IEC_Timer_0_DB_21".TON(pt := T#3S, et =>)
      Move(in := 1, out1 => "MODBUS DB"."STEP")
   END_RUNG
   RUNG wire#powerrail
      { S7_Templates := "SrcType := Int" } EQ_Contact(in1 := "MODBUS DB"."STEP", in2 := 14)
      Contact( "MODBUS DB".VFD_7.READ.BUSY )
   END_RUNG wire#w1
   // the same network as SCL:
   "IEC_Timer_0_DB_21".TON(IN := (("MODBUS DB"."STEP" = 13) AND "MODBUS DB".VFD_7.WRITE.BUSY) OR (("MODBUS DB"."STEP" = 14) AND "MODBUS DB".VFD_7.READ.BUSY),
                           PT := T#3S);
   IF "IEC_Timer_0_DB_21".Q THEN "MODBUS DB"."STEP" := 1; END_IF;
END_REGION
END_ORGANIZATION_BLOCK

DATA_BLOCK "SCALE AO_DB"   // DB171
// stored: InstanceOfName SCALE AO, InstanceOfType FB
"SCALE AO"
BEGIN
END_DATA_BLOCK

DATA_BLOCK "SCALE_DB"   // DB189
// stored: InstanceOfName SCALE, InstanceOfType FB
"SCALE"
BEGIN
END_DATA_BLOCK

DATA_BLOCK "SCALE_DB_1"   // DB190
// stored: InstanceOfName SCALE, InstanceOfType FB
"SCALE"
BEGIN
END_DATA_BLOCK

DATA_BLOCK "SCALE_DB_2"   // DB191
// stored: InstanceOfName SCALE, InstanceOfType FB
"SCALE"
BEGIN
END_DATA_BLOCK

DATA_BLOCK "SCALE_DB_3"   // DB192
// stored: InstanceOfName SCALE, InstanceOfType FB
"SCALE"
BEGIN
END_DATA_BLOCK

DATA_BLOCK "CONDUCTIVITY INDICATOR CUM TRANSMITTER_302"   // DB10
// stored: InstanceOfName SCALE, InstanceOfType FB
"SCALE"
BEGIN
END_DATA_BLOCK

DATA_BLOCK "CONDUCTIVITY INDICATOR CUM TRANSMITTER_401"   // DB13
// stored: InstanceOfName SCALE, InstanceOfType FB
"SCALE"
BEGIN
END_DATA_BLOCK

DATA_BLOCK "CONDUCTIVITY INDUCTOR CUM TRANSMITTER_301"   // DB7
// stored: InstanceOfName SCALE, InstanceOfType FB
"SCALE"
BEGIN
END_DATA_BLOCK

DATA_BLOCK "CONFUCTIVITY INDICATOR CUM TRANSMITTER_402"   // DB14
// stored: InstanceOfName SCALE, InstanceOfType FB
"SCALE"
BEGIN
END_DATA_BLOCK

DATA_BLOCK "FLOW INDICATOR TOTALOZER_501"   // DB17
// stored: InstanceOfName SCALE, InstanceOfType FB
"SCALE"
BEGIN
END_DATA_BLOCK

DATA_BLOCK "FLOW INDICATOR TRANSMITTER_502"   // DB19
// stored: InstanceOfName SCALE, InstanceOfType FB
"SCALE"
BEGIN
END_DATA_BLOCK

DATA_BLOCK "FLOW INDICATOR TRANSMITTER_503"   // DB30
// stored: InstanceOfName SCALE, InstanceOfType FB
"SCALE"
BEGIN
END_DATA_BLOCK

DATA_BLOCK "FLOW INDICATOR TRANSMITTER_504"   // DB31
// stored: InstanceOfName SCALE, InstanceOfType FB
"SCALE"
BEGIN
END_DATA_BLOCK

DATA_BLOCK "FLOW INDICATOR TRANSMITTER_505"   // DB32
// stored: InstanceOfName SCALE, InstanceOfType FB
"SCALE"
BEGIN
END_DATA_BLOCK

DATA_BLOCK "FLOW INDICATOR TRANSMITTER_506"   // DB33
// stored: InstanceOfName SCALE, InstanceOfType FB
"SCALE"
BEGIN
END_DATA_BLOCK

DATA_BLOCK "FLOW INDICATOR TRANSMITTER_507"   // DB34
// stored: InstanceOfName SCALE, InstanceOfType FB
"SCALE"
BEGIN
END_DATA_BLOCK

DATA_BLOCK "FLOW INDICATOR TRANSMITTER_508"   // DB35
// stored: InstanceOfName SCALE, InstanceOfType FB
"SCALE"
BEGIN
END_DATA_BLOCK

DATA_BLOCK "LEVEL TRANSMITTER_401"   // DB11
// stored: InstanceOfName SCALE, InstanceOfType FB
"SCALE"
BEGIN
END_DATA_BLOCK

DATA_BLOCK "LEVEL TRANSMITTER_501"   // DB16
// stored: InstanceOfName SCALE, InstanceOfType FB
"SCALE"
BEGIN
END_DATA_BLOCK

DATA_BLOCK "LEVEL TRANSMITTER_502"   // DB29
// stored: InstanceOfName SCALE, InstanceOfType FB
"SCALE"
BEGIN
END_DATA_BLOCK

DATA_BLOCK "OXIDATION REDUCTION POTENTIO_METER 301"   // DB6
// stored: InstanceOfName SCALE, InstanceOfType FB
"SCALE"
BEGIN
END_DATA_BLOCK

DATA_BLOCK "PH INDICATOR CUM TRANSMITTER_301"   // DB8
// stored: InstanceOfName SCALE, InstanceOfType FB
"SCALE"
BEGIN
END_DATA_BLOCK

DATA_BLOCK "PH INDICATOR CUM TRANSMITTER_302"   // DB9
// stored: InstanceOfName SCALE, InstanceOfType FB
"SCALE"
BEGIN
END_DATA_BLOCK

DATA_BLOCK "PH INDICATOR CUM TRANSMITTER_401"   // DB12
// stored: InstanceOfName SCALE, InstanceOfType FB
"SCALE"
BEGIN
END_DATA_BLOCK

DATA_BLOCK "PH INDICATOR CUM TRANSMITTER_402"   // DB15
// stored: InstanceOfName SCALE, InstanceOfType FB
"SCALE"
BEGIN
END_DATA_BLOCK

DATA_BLOCK "PH INDICATOR CUM TRANSMITTER_501"   // DB25
// stored: InstanceOfName SCALE, InstanceOfType FB
"SCALE"
BEGIN
END_DATA_BLOCK

DATA_BLOCK "PH INDICATOR CUM TRANSMITTER_502"   // DB26
// stored: InstanceOfName SCALE, InstanceOfType FB
"SCALE"
BEGIN
END_DATA_BLOCK

DATA_BLOCK "PRESSURE TRANSMITTER_501"   // DB18
// stored: InstanceOfName SCALE, InstanceOfType FB
"SCALE"
BEGIN
END_DATA_BLOCK

DATA_BLOCK "PRESSURE TRANSMITTER_502"   // DB20
// stored: InstanceOfName SCALE, InstanceOfType FB
"SCALE"
BEGIN
END_DATA_BLOCK

DATA_BLOCK "PRESSURE TRANSMITTER_503"   // DB21
// stored: InstanceOfName SCALE, InstanceOfType FB
"SCALE"
BEGIN
END_DATA_BLOCK

DATA_BLOCK "PRESSURE TRANSMITTER_504"   // DB22
// stored: InstanceOfName SCALE, InstanceOfType FB
"SCALE"
BEGIN
END_DATA_BLOCK

DATA_BLOCK "PRESSURE TRANSMITTER_505"   // DB23
// stored: InstanceOfName SCALE, InstanceOfType FB
"SCALE"
BEGIN
END_DATA_BLOCK

DATA_BLOCK "PRESSURE TRANSMITTER_506"   // DB24
// stored: InstanceOfName SCALE, InstanceOfType FB
"SCALE"
BEGIN
END_DATA_BLOCK

DATA_BLOCK "RESISTIVITY CUM TRANSMITTER_501"   // DB27
// stored: InstanceOfName SCALE, InstanceOfType FB
"SCALE"
BEGIN
END_DATA_BLOCK

DATA_BLOCK "RESISTIVITY CUM TRANSMITTER_502"   // DB28
// stored: InstanceOfName SCALE, InstanceOfType FB
"SCALE"
BEGIN
END_DATA_BLOCK

DATA_BLOCK "ABFV 501_FLUSH"   // DB206
// stored: InstanceOfName FLUSHING VALVE, InstanceOfType FB
"FLUSHING VALVE"
   // VAR_INPUT
   //    "SUBOUTPUT VALVE" : Bool;
   //    "OPEN FEEDBACK" : Bool;
   //    "CLOSE FEEDBACK" : Bool;
   // END_VAR
   // VAR_OUTPUT
   //    "OPEN OUTPUT VAVLE" : Bool;
   //    "CLOSE OUTPUT VAVLE" : Bool;
   // END_VAR
   // VAR
   //    TIMER_1 { S7_SetPoint := 'True'} : TON_TIME;
   //    "TIMER" { S7_SetPoint := 'True'} : TON_TIME;
   // END_VAR
BEGIN
END_DATA_BLOCK

DATA_BLOCK "ABFV 502_FLUSH"   // DB207
// stored: InstanceOfName FLUSHING VALVE, InstanceOfType FB
"FLUSHING VALVE"
   // VAR_INPUT
   //    "SUBOUTPUT VALVE" : Bool;
   //    "OPEN FEEDBACK" : Bool;
   //    "CLOSE FEEDBACK" : Bool;
   // END_VAR
   // VAR_OUTPUT
   //    "OPEN OUTPUT VAVLE" : Bool;
   //    "CLOSE OUTPUT VAVLE" : Bool;
   // END_VAR
   // VAR
   //    TIMER_1 { S7_SetPoint := 'True'} : TON_TIME;
   //    "TIMER" { S7_SetPoint := 'True'} : TON_TIME;
   // END_VAR
BEGIN
END_DATA_BLOCK

DATA_BLOCK "ABV 301_FLUSH"   // DB64
// stored: InstanceOfName FLUSHING VALVE, InstanceOfType FB
"FLUSHING VALVE"
   // VAR_INPUT
   //    "SUBOUTPUT VALVE" : Bool;
   //    "OPEN FEEDBACK" : Bool;
   //    "CLOSE FEEDBACK" : Bool;
   // END_VAR
   // VAR_OUTPUT
   //    "OPEN OUTPUT VAVLE" : Bool;
   //    "CLOSE OUTPUT VAVLE" : Bool;
   // END_VAR
   // VAR
   //    TIMER_1 { S7_SetPoint := 'True'} : TON_TIME;
   //    "TIMER" { S7_SetPoint := 'True'} : TON_TIME;
   // END_VAR
BEGIN
END_DATA_BLOCK

DATA_BLOCK "ABV 302_FLUSH"   // DB65
// stored: InstanceOfName FLUSHING VALVE, InstanceOfType FB
"FLUSHING VALVE"
   // VAR_INPUT
   //    "SUBOUTPUT VALVE" : Bool;
   //    "OPEN FEEDBACK" : Bool;
   //    "CLOSE FEEDBACK" : Bool;
   // END_VAR
   // VAR_OUTPUT
   //    "OPEN OUTPUT VAVLE" : Bool;
   //    "CLOSE OUTPUT VAVLE" : Bool;
   // END_VAR
   // VAR
   //    TIMER_1 { S7_SetPoint := 'True'} : TON_TIME;
   //    "TIMER" { S7_SetPoint := 'True'} : TON_TIME;
   // END_VAR
BEGIN
END_DATA_BLOCK

DATA_BLOCK "AGLV-301_FLUSH"   // DB66
// stored: InstanceOfName FLUSHING VALVE, InstanceOfType FB
"FLUSHING VALVE"
   // VAR_INPUT
   //    "SUBOUTPUT VALVE" : Bool;
   //    "OPEN FEEDBACK" : Bool;
   //    "CLOSE FEEDBACK" : Bool;
   // END_VAR
   // VAR_OUTPUT
   //    "OPEN OUTPUT VAVLE" : Bool;
   //    "CLOSE OUTPUT VAVLE" : Bool;
   // END_VAR
   // VAR
   //    TIMER_1 { S7_SetPoint := 'True'} : TON_TIME;
   //    "TIMER" { S7_SetPoint := 'True'} : TON_TIME;
   // END_VAR
BEGIN
END_DATA_BLOCK

DATA_BLOCK "AGLV-302_FLUSH"   // DB67
// stored: InstanceOfName FLUSHING VALVE, InstanceOfType FB
"FLUSHING VALVE"
   // VAR_INPUT
   //    "SUBOUTPUT VALVE" : Bool;
   //    "OPEN FEEDBACK" : Bool;
   //    "CLOSE FEEDBACK" : Bool;
   // END_VAR
   // VAR_OUTPUT
   //    "OPEN OUTPUT VAVLE" : Bool;
   //    "CLOSE OUTPUT VAVLE" : Bool;
   // END_VAR
   // VAR
   //    TIMER_1 { S7_SetPoint := 'True'} : TON_TIME;
   //    "TIMER" { S7_SetPoint := 'True'} : TON_TIME;
   // END_VAR
BEGIN
END_DATA_BLOCK

DATA_BLOCK "AGLV-401_FLUSH"   // DB68
// stored: InstanceOfName FLUSHING VALVE, InstanceOfType FB
"FLUSHING VALVE"
   // VAR_INPUT
   //    "SUBOUTPUT VALVE" : Bool;
   //    "OPEN FEEDBACK" : Bool;
   //    "CLOSE FEEDBACK" : Bool;
   // END_VAR
   // VAR_OUTPUT
   //    "OPEN OUTPUT VAVLE" : Bool;
   //    "CLOSE OUTPUT VAVLE" : Bool;
   // END_VAR
   // VAR
   //    TIMER_1 { S7_SetPoint := 'True'} : TON_TIME;
   //    "TIMER" { S7_SetPoint := 'True'} : TON_TIME;
   // END_VAR
BEGIN
END_DATA_BLOCK

DATA_BLOCK "AGLV-402_FLUSH"   // DB69
// stored: InstanceOfName FLUSHING VALVE, InstanceOfType FB
"FLUSHING VALVE"
   // VAR_INPUT
   //    "SUBOUTPUT VALVE" : Bool;
   //    "OPEN FEEDBACK" : Bool;
   //    "CLOSE FEEDBACK" : Bool;
   // END_VAR
   // VAR_OUTPUT
   //    "OPEN OUTPUT VAVLE" : Bool;
   //    "CLOSE OUTPUT VAVLE" : Bool;
   // END_VAR
   // VAR
   //    TIMER_1 { S7_SetPoint := 'True'} : TON_TIME;
   //    "TIMER" { S7_SetPoint := 'True'} : TON_TIME;
   // END_VAR
BEGIN
END_DATA_BLOCK

DATA_BLOCK "TIMING_MIN_DB_5"   // DB241
// stored: InstanceOfName TIMING_MIN, InstanceOfType FB
"TIMING_MIN"
   // VAR_INPUT
   //    "SET TIME" : Int;
   //    RESET : Bool;
   //    INPUT : Bool;
   // END_VAR
   // VAR_OUTPUT
   //    "PRESENT VALUE OF TIME" : Int;
   //    DONE : Bool;
   // END_VAR
   // VAR
   //    "TIMER 1" { S7_SetPoint := 'True'} : IEC_TIMER;
   // END_VAR
   // VAR RETAIN
   //    "COUNTER1 1" { S7_SetPoint := 'True'} : IEC_COUNTER;
   // END_VAR
BEGIN
END_DATA_BLOCK

DATA_BLOCK "TIMING_MIN_DB_6"   // DB242
// stored: InstanceOfName TIMING_MIN, InstanceOfType FB
"TIMING_MIN"
   // VAR_INPUT
   //    "SET TIME" : Int;
   //    RESET : Bool;
   //    INPUT : Bool;
   // END_VAR
   // VAR_OUTPUT
   //    "PRESENT VALUE OF TIME" : Int;
   //    DONE : Bool;
   // END_VAR
   // VAR
   //    "TIMER 1" { S7_SetPoint := 'True'} : IEC_TIMER;
   // END_VAR
   // VAR RETAIN
   //    "COUNTER1 1" { S7_SetPoint := 'True'} : IEC_COUNTER;
   // END_VAR
BEGIN
END_DATA_BLOCK

DATA_BLOCK "TIMING_MIN_DB_7"   // DB240
// stored: InstanceOfName TIMING_MIN, InstanceOfType FB
"TIMING_MIN"
   // VAR_INPUT
   //    "SET TIME" : Int;
   //    RESET : Bool;
   //    INPUT : Bool;
   // END_VAR
   // VAR_OUTPUT
   //    "PRESENT VALUE OF TIME" : Int;
   //    DONE : Bool;
   // END_VAR
   // VAR
   //    "TIMER 1" { S7_SetPoint := 'True'} : IEC_TIMER;
   // END_VAR
   // VAR RETAIN
   //    "COUNTER1 1" { S7_SetPoint := 'True'} : IEC_COUNTER;
   // END_VAR
BEGIN
END_DATA_BLOCK

DATA_BLOCK "TIMING_MIN_DB_8"   // DB245
// stored: InstanceOfName TIMING_MIN, InstanceOfType FB
"TIMING_MIN"
   // VAR_INPUT
   //    "SET TIME" : Int;
   //    RESET : Bool;
   //    INPUT : Bool;
   // END_VAR
   // VAR_OUTPUT
   //    "PRESENT VALUE OF TIME" : Int;
   //    DONE : Bool;
   // END_VAR
   // VAR
   //    "TIMER 1" { S7_SetPoint := 'True'} : IEC_TIMER;
   // END_VAR
   // VAR RETAIN
   //    "COUNTER1 1" { S7_SetPoint := 'True'} : IEC_COUNTER;
   // END_VAR
BEGIN
END_DATA_BLOCK

DATA_BLOCK "TIMING_MIN_DB_10"   // DB40
// stored: InstanceOfName TIMING_MIN, InstanceOfType FB
"TIMING_MIN"
   // VAR_INPUT
   //    "SET TIME" : Int;
   //    RESET : Bool;
   //    INPUT : Bool;
   // END_VAR
   // VAR_OUTPUT
   //    "PRESENT VALUE OF TIME" : Int;
   //    DONE : Bool;
   // END_VAR
   // VAR
   //    "TIMER 1" { S7_SetPoint := 'True'} : IEC_TIMER;
   // END_VAR
   // VAR RETAIN
   //    "COUNTER1 1" { S7_SetPoint := 'True'} : IEC_COUNTER;
   // END_VAR
BEGIN
END_DATA_BLOCK

DATA_BLOCK "TIMING_MIN_DB_9"   // DB39
// stored: InstanceOfName TIMING_MIN, InstanceOfType FB
"TIMING_MIN"
   // VAR_INPUT
   //    "SET TIME" : Int;
   //    RESET : Bool;
   //    INPUT : Bool;
   // END_VAR
   // VAR_OUTPUT
   //    "PRESENT VALUE OF TIME" : Int;
   //    DONE : Bool;
   // END_VAR
   // VAR
   //    "TIMER 1" { S7_SetPoint := 'True'} : IEC_TIMER;
   // END_VAR
   // VAR RETAIN
   //    "COUNTER1 1" { S7_SetPoint := 'True'} : IEC_COUNTER;
   // END_VAR
BEGIN
END_DATA_BLOCK

DATA_BLOCK "TIMING_MIN_DB"   // DB93
// stored: InstanceOfName TIMING_MIN, InstanceOfType FB
"TIMING_MIN"
   // VAR_INPUT
   //    "SET TIME" : Int;
   //    RESET : Bool;
   //    INPUT : Bool;
   // END_VAR
   // VAR_OUTPUT
   //    "PRESENT VALUE OF TIME" : Int;
   //    DONE : Bool;
   // END_VAR
   // VAR
   //    "TIMER 1" { S7_SetPoint := 'True'} : IEC_TIMER;
   // END_VAR
   // VAR RETAIN
   //    "COUNTER1 1" { S7_SetPoint := 'True'} : IEC_COUNTER;
   // END_VAR
BEGIN
END_DATA_BLOCK

DATA_BLOCK "TIMING_MIN_DB_1"   // DB100
// stored: InstanceOfName TIMING_MIN, InstanceOfType FB
"TIMING_MIN"
   // VAR_INPUT
   //    "SET TIME" : Int;
   //    RESET : Bool;
   //    INPUT : Bool;
   // END_VAR
   // VAR_OUTPUT
   //    "PRESENT VALUE OF TIME" : Int;
   //    DONE : Bool;
   // END_VAR
   // VAR
   //    "TIMER 1" { S7_SetPoint := 'True'} : IEC_TIMER;
   // END_VAR
   // VAR RETAIN
   //    "COUNTER1 1" { S7_SetPoint := 'True'} : IEC_COUNTER;
   // END_VAR
BEGIN
END_DATA_BLOCK

DATA_BLOCK "TIMING_MIN_DB_2"   // DB147
// stored: InstanceOfName TIMING_MIN, InstanceOfType FB
"TIMING_MIN"
   // VAR_INPUT
   //    "SET TIME" : Int;
   //    RESET : Bool;
   //    INPUT : Bool;
   // END_VAR
   // VAR_OUTPUT
   //    "PRESENT VALUE OF TIME" : Int;
   //    DONE : Bool;
   // END_VAR
   // VAR
   //    "TIMER 1" { S7_SetPoint := 'True'} : IEC_TIMER;
   // END_VAR
   // VAR RETAIN
   //    "COUNTER1 1" { S7_SetPoint := 'True'} : IEC_COUNTER;
   // END_VAR
BEGIN
END_DATA_BLOCK

DATA_BLOCK "TIMING_MIN_DB_3"   // DB101
// stored: InstanceOfName TIMING_MIN, InstanceOfType FB
"TIMING_MIN"
   // VAR_INPUT
   //    "SET TIME" : Int;
   //    RESET : Bool;
   //    INPUT : Bool;
   // END_VAR
   // VAR_OUTPUT
   //    "PRESENT VALUE OF TIME" : Int;
   //    DONE : Bool;
   // END_VAR
   // VAR
   //    "TIMER 1" { S7_SetPoint := 'True'} : IEC_TIMER;
   // END_VAR
   // VAR RETAIN
   //    "COUNTER1 1" { S7_SetPoint := 'True'} : IEC_COUNTER;
   // END_VAR
BEGIN
END_DATA_BLOCK

DATA_BLOCK "TIMING_MIN_DB_4"   // DB95
// stored: InstanceOfName TIMING_MIN, InstanceOfType FB
"TIMING_MIN"
   // VAR_INPUT
   //    "SET TIME" : Int;
   //    RESET : Bool;
   //    INPUT : Bool;
   // END_VAR
   // VAR_OUTPUT
   //    "PRESENT VALUE OF TIME" : Int;
   //    DONE : Bool;
   // END_VAR
   // VAR
   //    "TIMER 1" { S7_SetPoint := 'True'} : IEC_TIMER;
   // END_VAR
   // VAR RETAIN
   //    "COUNTER1 1" { S7_SetPoint := 'True'} : IEC_COUNTER;
   // END_VAR
BEGIN
END_DATA_BLOCK

DATA_BLOCK "TIMING_SECS_DB"   // DB89
// stored: InstanceOfName TIMING_SECS, InstanceOfType FB
"TIMING_SECS"
BEGIN
END_DATA_BLOCK

DATA_BLOCK "TIMING_SECS_DB_1"   // DB90
// stored: InstanceOfName TIMING_SECS, InstanceOfType FB
"TIMING_SECS"
BEGIN
END_DATA_BLOCK

DATA_BLOCK "TIMING_SECS_DB_10"   // DB148
// stored: InstanceOfName TIMING_SECS, InstanceOfType FB
"TIMING_SECS"
BEGIN
END_DATA_BLOCK

DATA_BLOCK "TIMING_SECS_DB_11"   // DB149
// stored: InstanceOfName TIMING_SECS, InstanceOfType FB
"TIMING_SECS"
BEGIN
END_DATA_BLOCK

DATA_BLOCK "TIMING_SECS_DB_12"   // DB115
// stored: InstanceOfName TIMING_SECS, InstanceOfType FB
"TIMING_SECS"
BEGIN
END_DATA_BLOCK

DATA_BLOCK "TIMING_SECS_DB_13"   // DB150
// stored: InstanceOfName TIMING_SECS, InstanceOfType FB
"TIMING_SECS"
BEGIN
END_DATA_BLOCK

DATA_BLOCK "TIMING_SECS_DB_14"   // DB151
// stored: InstanceOfName TIMING_SECS, InstanceOfType FB
"TIMING_SECS"
BEGIN
END_DATA_BLOCK

DATA_BLOCK "TIMING_SECS_DB_15"   // DB152
// stored: InstanceOfName TIMING_SECS, InstanceOfType FB
"TIMING_SECS"
BEGIN
END_DATA_BLOCK

DATA_BLOCK "TIMING_SECS_DB_16"   // DB118
// stored: InstanceOfName TIMING_SECS, InstanceOfType FB
"TIMING_SECS"
BEGIN
END_DATA_BLOCK

DATA_BLOCK "TIMING_SECS_DB_17"   // DB119
// stored: InstanceOfName TIMING_SECS, InstanceOfType FB
"TIMING_SECS"
BEGIN
END_DATA_BLOCK

DATA_BLOCK "TIMING_SECS_DB_18"   // DB157
// stored: InstanceOfName TIMING_SECS, InstanceOfType FB
"TIMING_SECS"
BEGIN
END_DATA_BLOCK

DATA_BLOCK "TIMING_SECS_DB_19"   // DB154
// stored: InstanceOfName TIMING_SECS, InstanceOfType FB
"TIMING_SECS"
BEGIN
END_DATA_BLOCK

DATA_BLOCK "TIMING_SECS_DB_2"   // DB91
// stored: InstanceOfName TIMING_SECS, InstanceOfType FB
"TIMING_SECS"
BEGIN
END_DATA_BLOCK

DATA_BLOCK "TIMING_SECS_DB_20"   // DB155
// stored: InstanceOfName TIMING_SECS, InstanceOfType FB
"TIMING_SECS"
BEGIN
END_DATA_BLOCK

DATA_BLOCK "TIMING_SECS_DB_21"   // DB156
// stored: InstanceOfName TIMING_SECS, InstanceOfType FB
"TIMING_SECS"
BEGIN
END_DATA_BLOCK

DATA_BLOCK "TIMING_SECS_DB_22"   // DB159
// stored: InstanceOfName TIMING_SECS, InstanceOfType FB
"TIMING_SECS"
BEGIN
END_DATA_BLOCK

DATA_BLOCK "TIMING_SECS_DB_23"   // DB158
// stored: InstanceOfName TIMING_SECS, InstanceOfType FB
"TIMING_SECS"
BEGIN
END_DATA_BLOCK

DATA_BLOCK "TIMING_SECS_DB_24"   // DB120
// stored: InstanceOfName TIMING_SECS, InstanceOfType FB
"TIMING_SECS"
BEGIN
END_DATA_BLOCK

DATA_BLOCK "TIMING_SECS_DB_25"   // DB168
// stored: InstanceOfName TIMING_SECS, InstanceOfType FB
"TIMING_SECS"
BEGIN
END_DATA_BLOCK

DATA_BLOCK "TIMING_SECS_DB_26"   // DB163
// stored: InstanceOfName TIMING_SECS, InstanceOfType FB
"TIMING_SECS"
BEGIN
END_DATA_BLOCK

DATA_BLOCK "TIMING_SECS_DB_27"   // DB167
// stored: InstanceOfName TIMING_SECS, InstanceOfType FB
"TIMING_SECS"
BEGIN
END_DATA_BLOCK

DATA_BLOCK "TIMING_SECS_DB_28"   // DB166
// stored: InstanceOfName TIMING_SECS, InstanceOfType FB
"TIMING_SECS"
BEGIN
END_DATA_BLOCK

DATA_BLOCK "TIMING_SECS_DB_29"   // DB161
// stored: InstanceOfName TIMING_SECS, InstanceOfType FB
"TIMING_SECS"
BEGIN
END_DATA_BLOCK

DATA_BLOCK "TIMING_SECS_DB_3"   // DB92
// stored: InstanceOfName TIMING_SECS, InstanceOfType FB
"TIMING_SECS"
BEGIN
END_DATA_BLOCK

DATA_BLOCK "TIMING_SECS_DB_30"   // DB160
// stored: InstanceOfName TIMING_SECS, InstanceOfType FB
"TIMING_SECS"
BEGIN
END_DATA_BLOCK

DATA_BLOCK "TIMING_SECS_DB_31"   // DB162
// stored: InstanceOfName TIMING_SECS, InstanceOfType FB
"TIMING_SECS"
BEGIN
END_DATA_BLOCK

DATA_BLOCK "TIMING_SECS_DB_32"   // DB164
// stored: InstanceOfName TIMING_SECS, InstanceOfType FB
"TIMING_SECS"
BEGIN
END_DATA_BLOCK

DATA_BLOCK "TIMING_SECS_DB_33"   // DB165
// stored: InstanceOfName TIMING_SECS, InstanceOfType FB
"TIMING_SECS"
BEGIN
END_DATA_BLOCK

DATA_BLOCK "TIMING_SECS_DB_34"   // DB169
// stored: InstanceOfName TIMING_SECS, InstanceOfType FB
"TIMING_SECS"
BEGIN
END_DATA_BLOCK

DATA_BLOCK "TIMING_SECS_DB_35"   // DB141
// stored: InstanceOfName TIMING_SECS, InstanceOfType FB
"TIMING_SECS"
BEGIN
END_DATA_BLOCK

DATA_BLOCK "TIMING_SECS_DB_4"   // DB146
// stored: InstanceOfName TIMING_SECS, InstanceOfType FB
"TIMING_SECS"
BEGIN
END_DATA_BLOCK

DATA_BLOCK "TIMING_SECS_DB_5"   // DB145
// stored: InstanceOfName TIMING_SECS, InstanceOfType FB
"TIMING_SECS"
BEGIN
END_DATA_BLOCK

DATA_BLOCK "TIMING_SECS_DB_6"   // DB144
// stored: InstanceOfName TIMING_SECS, InstanceOfType FB
"TIMING_SECS"
BEGIN
END_DATA_BLOCK

DATA_BLOCK "TIMING_SECS_DB_7"   // DB117
// stored: InstanceOfName TIMING_SECS, InstanceOfType FB
"TIMING_SECS"
BEGIN
END_DATA_BLOCK

DATA_BLOCK "TIMING_SECS_DB_8"   // DB114
// stored: InstanceOfName TIMING_SECS, InstanceOfType FB
"TIMING_SECS"
BEGIN
END_DATA_BLOCK

DATA_BLOCK "TIMING_SECS_DB_9"   // DB153
// stored: InstanceOfName TIMING_SECS, InstanceOfType FB
"TIMING_SECS"
BEGIN
END_DATA_BLOCK

DATA_BLOCK "IEC_Counter_0_DB"   // DB201
{ S7_Optimized_Access := 'TRUE' }
// stored: InstanceOfName IEC_COUNTER, OfSystemLibElement IEC_COUNTER, OfSystemLibVersion 1.0
"IEC_COUNTER"
   // VAR RETAIN
   //    CU : Bool;
   //    CD : Bool;
   //    R : Bool;
   //    LD : Bool;
   //    QU : Bool;
   //    QD : Bool;
   //    PV : Int;
   //    CV : Int;
   // END_VAR
BEGIN
END_DATA_BLOCK

DATA_BLOCK "IEC_Counter_0_DB_1"   // DB203
{ S7_Optimized_Access := 'TRUE' }
// stored: InstanceOfName IEC_COUNTER, OfSystemLibElement IEC_COUNTER, OfSystemLibVersion 1.0
"IEC_COUNTER"
   // VAR RETAIN
   //    CU : Bool;
   //    CD : Bool;
   //    R : Bool;
   //    LD : Bool;
   //    QU : Bool;
   //    QD : Bool;
   //    PV : Int;
   //    CV : Int;
   // END_VAR
BEGIN
END_DATA_BLOCK

DATA_BLOCK "IEC_Counter_0_DB_4"   // DB212
{ S7_Optimized_Access := 'TRUE' }
// stored: InstanceOfName IEC_COUNTER, OfSystemLibElement IEC_COUNTER, OfSystemLibVersion 1.0
"IEC_COUNTER"
   // VAR RETAIN
   //    CU : Bool;
   //    CD : Bool;
   //    R : Bool;
   //    LD : Bool;
   //    QU : Bool;
   //    QD : Bool;
   //    PV : Int;
   //    CV : Int;
   // END_VAR
BEGIN
END_DATA_BLOCK

DATA_BLOCK "IEC_Counter_0_DB_5"   // DB214
{ S7_Optimized_Access := 'TRUE' }
// stored: InstanceOfName IEC_COUNTER, OfSystemLibElement IEC_COUNTER, OfSystemLibVersion 1.0
"IEC_COUNTER"
   // VAR RETAIN
   //    CU : Bool;
   //    CD : Bool;
   //    R : Bool;
   //    LD : Bool;
   //    QU : Bool;
   //    QD : Bool;
   //    PV : Int;
   //    CV : Int;
   // END_VAR
BEGIN
END_DATA_BLOCK

DATA_BLOCK "IEC_Counter_0_DB_8"   // DB223
{ S7_Optimized_Access := 'TRUE' }
// stored: InstanceOfName IEC_COUNTER, OfSystemLibElement IEC_COUNTER, OfSystemLibVersion 1.0
"IEC_COUNTER"
   // VAR RETAIN
   //    CU : Bool;
   //    CD : Bool;
   //    R : Bool;
   //    LD : Bool;
   //    QU : Bool;
   //    QD : Bool;
   //    PV : Int;
   //    CV : Int;
   // END_VAR
BEGIN
END_DATA_BLOCK

DATA_BLOCK "IEC_Timer_0_DB"   // DB38
{ S7_Optimized_Access := 'TRUE' }
// stored: InstanceOfName IEC_TIMER, OfSystemLibElement IEC_TIMER, OfSystemLibVersion 1.0
"IEC_TIMER"
   // VAR
   //    PT : Time;
   //    ET { ExternalWritable := 'False'} : Time;
   //    IN : Bool;
   //    Q { ExternalWritable := 'False'} : Bool;
   // END_VAR
BEGIN
END_DATA_BLOCK

DATA_BLOCK "IEC_Timer_0_DB_1"   // DB41
{ S7_Optimized_Access := 'TRUE' }
// stored: InstanceOfName IEC_TIMER, OfSystemLibElement IEC_TIMER, OfSystemLibVersion 1.0
"IEC_TIMER"
   // VAR
   //    PT : Time;
   //    ET { ExternalWritable := 'False'} : Time;
   //    IN : Bool;
   //    Q { ExternalWritable := 'False'} : Bool;
   // END_VAR
BEGIN
END_DATA_BLOCK

DATA_BLOCK "IEC_Timer_0_DB_10"   // DB50
{ S7_Optimized_Access := 'TRUE' }
// stored: InstanceOfName IEC_TIMER, OfSystemLibElement IEC_TIMER, OfSystemLibVersion 1.0
"IEC_TIMER"
   // VAR
   //    PT : Time;
   //    ET { ExternalWritable := 'False'} : Time;
   //    IN : Bool;
   //    Q { ExternalWritable := 'False'} : Bool;
   // END_VAR
BEGIN
END_DATA_BLOCK

DATA_BLOCK "IEC_Timer_0_DB_100"   // DB224
{ S7_Optimized_Access := 'TRUE' }
// stored: InstanceOfName IEC_TIMER, OfSystemLibElement IEC_TIMER, OfSystemLibVersion 1.0
"IEC_TIMER"
   // VAR
   //    PT : Time;
   //    ET { ExternalWritable := 'False'} : Time;
   //    IN : Bool;
   //    Q { ExternalWritable := 'False'} : Bool;
   // END_VAR
BEGIN
END_DATA_BLOCK

DATA_BLOCK "IEC_Timer_0_DB_101"   // DB225
{ S7_Optimized_Access := 'TRUE' }
// stored: InstanceOfName IEC_TIMER, OfSystemLibElement IEC_TIMER, OfSystemLibVersion 1.0
"IEC_TIMER"
   // VAR
   //    PT : Time;
   //    ET { ExternalWritable := 'False'} : Time;
   //    IN : Bool;
   //    Q { ExternalWritable := 'False'} : Bool;
   // END_VAR
BEGIN
END_DATA_BLOCK

DATA_BLOCK "IEC_Timer_0_DB_102"   // DB226
{ S7_Optimized_Access := 'TRUE' }
// stored: InstanceOfName IEC_TIMER, OfSystemLibElement IEC_TIMER, OfSystemLibVersion 1.0
"IEC_TIMER"
   // VAR
   //    PT : Time;
   //    ET { ExternalWritable := 'False'} : Time;
   //    IN : Bool;
   //    Q { ExternalWritable := 'False'} : Bool;
   // END_VAR
BEGIN
END_DATA_BLOCK

DATA_BLOCK "IEC_Timer_0_DB_103"   // DB227
{ S7_Optimized_Access := 'TRUE' }
// stored: InstanceOfName IEC_TIMER, OfSystemLibElement IEC_TIMER, OfSystemLibVersion 1.0
"IEC_TIMER"
   // VAR
   //    PT : Time;
   //    ET { ExternalWritable := 'False'} : Time;
   //    IN : Bool;
   //    Q { ExternalWritable := 'False'} : Bool;
   // END_VAR
BEGIN
END_DATA_BLOCK

DATA_BLOCK "IEC_Timer_0_DB_104"   // DB229
{ S7_Optimized_Access := 'TRUE' }
// stored: InstanceOfName IEC_TIMER, OfSystemLibElement IEC_TIMER, OfSystemLibVersion 1.0
"IEC_TIMER"
   // VAR
   //    PT : Time;
   //    ET { ExternalWritable := 'False'} : Time;
   //    IN : Bool;
   //    Q { ExternalWritable := 'False'} : Bool;
   // END_VAR
BEGIN
END_DATA_BLOCK

DATA_BLOCK "IEC_Timer_0_DB_105"   // DB230
{ S7_Optimized_Access := 'TRUE' }
// stored: InstanceOfName IEC_TIMER, OfSystemLibElement IEC_TIMER, OfSystemLibVersion 1.0
"IEC_TIMER"
   // VAR
   //    PT : Time;
   //    ET { ExternalWritable := 'False'} : Time;
   //    IN : Bool;
   //    Q { ExternalWritable := 'False'} : Bool;
   // END_VAR
BEGIN
END_DATA_BLOCK

DATA_BLOCK "IEC_Timer_0_DB_106"   // DB231
{ S7_Optimized_Access := 'TRUE' }
// stored: InstanceOfName IEC_TIMER, OfSystemLibElement IEC_TIMER, OfSystemLibVersion 1.0
"IEC_TIMER"
   // VAR
   //    PT : Time;
   //    ET { ExternalWritable := 'False'} : Time;
   //    IN : Bool;
   //    Q { ExternalWritable := 'False'} : Bool;
   // END_VAR
BEGIN
END_DATA_BLOCK

DATA_BLOCK "IEC_Timer_0_DB_107"   // DB232
{ S7_Optimized_Access := 'TRUE' }
// stored: InstanceOfName IEC_TIMER, OfSystemLibElement IEC_TIMER, OfSystemLibVersion 1.0
"IEC_TIMER"
   // VAR
   //    PT : Time;
   //    ET { ExternalWritable := 'False'} : Time;
   //    IN : Bool;
   //    Q { ExternalWritable := 'False'} : Bool;
   // END_VAR
BEGIN
END_DATA_BLOCK

DATA_BLOCK "IEC_Timer_0_DB_108"   // DB233
{ S7_Optimized_Access := 'TRUE' }
// stored: InstanceOfName IEC_TIMER, OfSystemLibElement IEC_TIMER, OfSystemLibVersion 1.0
"IEC_TIMER"
   // VAR
   //    PT : Time;
   //    ET { ExternalWritable := 'False'} : Time;
   //    IN : Bool;
   //    Q { ExternalWritable := 'False'} : Bool;
   // END_VAR
BEGIN
END_DATA_BLOCK

DATA_BLOCK "IEC_Timer_0_DB_109"   // DB234
{ S7_Optimized_Access := 'TRUE' }
// stored: InstanceOfName IEC_TIMER, OfSystemLibElement IEC_TIMER, OfSystemLibVersion 1.0
"IEC_TIMER"
   // VAR
   //    PT : Time;
   //    ET { ExternalWritable := 'False'} : Time;
   //    IN : Bool;
   //    Q { ExternalWritable := 'False'} : Bool;
   // END_VAR
BEGIN
END_DATA_BLOCK

DATA_BLOCK "IEC_Timer_0_DB_11"   // DB51
{ S7_Optimized_Access := 'TRUE' }
// stored: InstanceOfName IEC_TIMER, OfSystemLibElement IEC_TIMER, OfSystemLibVersion 1.0
"IEC_TIMER"
   // VAR
   //    PT : Time;
   //    ET { ExternalWritable := 'False'} : Time;
   //    IN : Bool;
   //    Q { ExternalWritable := 'False'} : Bool;
   // END_VAR
BEGIN
END_DATA_BLOCK

DATA_BLOCK "IEC_Timer_0_DB_110"   // DB235
{ S7_Optimized_Access := 'TRUE' }
// stored: InstanceOfName IEC_TIMER, OfSystemLibElement IEC_TIMER, OfSystemLibVersion 1.0
"IEC_TIMER"
   // VAR
   //    PT : Time;
   //    ET { ExternalWritable := 'False'} : Time;
   //    IN : Bool;
   //    Q { ExternalWritable := 'False'} : Bool;
   // END_VAR
BEGIN
END_DATA_BLOCK

DATA_BLOCK "IEC_Timer_0_DB_111"   // DB236
{ S7_Optimized_Access := 'TRUE' }
// stored: InstanceOfName IEC_TIMER, OfSystemLibElement IEC_TIMER, OfSystemLibVersion 1.0
"IEC_TIMER"
   // VAR
   //    PT : Time;
   //    ET { ExternalWritable := 'False'} : Time;
   //    IN : Bool;
   //    Q { ExternalWritable := 'False'} : Bool;
   // END_VAR
BEGIN
END_DATA_BLOCK

DATA_BLOCK "IEC_Timer_0_DB_112"   // DB238
{ S7_Optimized_Access := 'TRUE' }
// stored: InstanceOfName IEC_TIMER, OfSystemLibElement IEC_TIMER, OfSystemLibVersion 1.0
"IEC_TIMER"
   // VAR
   //    PT : Time;
   //    ET { ExternalWritable := 'False'} : Time;
   //    IN : Bool;
   //    Q { ExternalWritable := 'False'} : Bool;
   // END_VAR
BEGIN
END_DATA_BLOCK

DATA_BLOCK "IEC_Timer_0_DB_113"   // DB239
{ S7_Optimized_Access := 'TRUE' }
// stored: InstanceOfName IEC_TIMER, OfSystemLibElement IEC_TIMER, OfSystemLibVersion 1.0
"IEC_TIMER"
   // VAR
   //    PT : Time;
   //    ET { ExternalWritable := 'False'} : Time;
   //    IN : Bool;
   //    Q { ExternalWritable := 'False'} : Bool;
   // END_VAR
BEGIN
END_DATA_BLOCK

DATA_BLOCK "IEC_Timer_0_DB_114"   // DB243
{ S7_Optimized_Access := 'TRUE' }
// stored: InstanceOfName IEC_TIMER, OfSystemLibElement IEC_TIMER, OfSystemLibVersion 1.0
"IEC_TIMER"
   // VAR
   //    PT : Time;
   //    ET { ExternalWritable := 'False'} : Time;
   //    IN : Bool;
   //    Q { ExternalWritable := 'False'} : Bool;
   // END_VAR
BEGIN
END_DATA_BLOCK

DATA_BLOCK "IEC_Timer_0_DB_115"   // DB244
{ S7_Optimized_Access := 'TRUE' }
// stored: InstanceOfName IEC_TIMER, OfSystemLibElement IEC_TIMER, OfSystemLibVersion 1.0
"IEC_TIMER"
   // VAR
   //    PT : Time;
   //    ET { ExternalWritable := 'False'} : Time;
   //    IN : Bool;
   //    Q { ExternalWritable := 'False'} : Bool;
   // END_VAR
BEGIN
END_DATA_BLOCK

DATA_BLOCK "IEC_Timer_0_DB_116"   // DB246
{ S7_Optimized_Access := 'TRUE' }
// stored: InstanceOfName IEC_TIMER, OfSystemLibElement IEC_TIMER, OfSystemLibVersion 1.0
"IEC_TIMER"
   // VAR
   //    PT : Time;
   //    ET { ExternalWritable := 'False'} : Time;
   //    IN : Bool;
   //    Q { ExternalWritable := 'False'} : Bool;
   // END_VAR
BEGIN
END_DATA_BLOCK

DATA_BLOCK "IEC_Timer_0_DB_117"   // DB247
{ S7_Optimized_Access := 'TRUE' }
// stored: InstanceOfName IEC_TIMER, OfSystemLibElement IEC_TIMER, OfSystemLibVersion 1.0
"IEC_TIMER"
   // VAR
   //    PT : Time;
   //    ET { ExternalWritable := 'False'} : Time;
   //    IN : Bool;
   //    Q { ExternalWritable := 'False'} : Bool;
   // END_VAR
BEGIN
END_DATA_BLOCK

DATA_BLOCK "IEC_Timer_0_DB_118"   // DB248
{ S7_Optimized_Access := 'TRUE' }
// stored: InstanceOfName IEC_TIMER, OfSystemLibElement IEC_TIMER, OfSystemLibVersion 1.0
"IEC_TIMER"
   // VAR
   //    PT : Time;
   //    ET { ExternalWritable := 'False'} : Time;
   //    IN : Bool;
   //    Q { ExternalWritable := 'False'} : Bool;
   // END_VAR
BEGIN
END_DATA_BLOCK

DATA_BLOCK "IEC_Timer_0_DB_119"   // DB249
{ S7_Optimized_Access := 'TRUE' }
// stored: InstanceOfName IEC_TIMER, OfSystemLibElement IEC_TIMER, OfSystemLibVersion 1.0
"IEC_TIMER"
   // VAR
   //    PT : Time;
   //    ET { ExternalWritable := 'False'} : Time;
   //    IN : Bool;
   //    Q { ExternalWritable := 'False'} : Bool;
   // END_VAR
BEGIN
END_DATA_BLOCK

DATA_BLOCK "IEC_Timer_0_DB_12"   // DB52
{ S7_Optimized_Access := 'TRUE' }
// stored: InstanceOfName IEC_TIMER, OfSystemLibElement IEC_TIMER, OfSystemLibVersion 1.0
"IEC_TIMER"
   // VAR
   //    PT : Time;
   //    ET { ExternalWritable := 'False'} : Time;
   //    IN : Bool;
   //    Q { ExternalWritable := 'False'} : Bool;
   // END_VAR
BEGIN
END_DATA_BLOCK

DATA_BLOCK "IEC_Timer_0_DB_120"   // DB250
{ S7_Optimized_Access := 'TRUE' }
// stored: InstanceOfName IEC_TIMER, OfSystemLibElement IEC_TIMER, OfSystemLibVersion 1.0
"IEC_TIMER"
   // VAR
   //    PT : Time;
   //    ET { ExternalWritable := 'False'} : Time;
   //    IN : Bool;
   //    Q { ExternalWritable := 'False'} : Bool;
   // END_VAR
BEGIN
END_DATA_BLOCK

DATA_BLOCK "IEC_Timer_0_DB_121"   // DB251
{ S7_Optimized_Access := 'TRUE' }
// stored: InstanceOfName IEC_TIMER, OfSystemLibElement IEC_TIMER, OfSystemLibVersion 1.0
"IEC_TIMER"
   // VAR
   //    PT : Time;
   //    ET { ExternalWritable := 'False'} : Time;
   //    IN : Bool;
   //    Q { ExternalWritable := 'False'} : Bool;
   // END_VAR
BEGIN
END_DATA_BLOCK

DATA_BLOCK "IEC_Timer_0_DB_122"   // DB252
{ S7_Optimized_Access := 'TRUE' }
// stored: InstanceOfName IEC_TIMER, OfSystemLibElement IEC_TIMER, OfSystemLibVersion 1.0
"IEC_TIMER"
   // VAR
   //    PT : Time;
   //    ET { ExternalWritable := 'False'} : Time;
   //    IN : Bool;
   //    Q { ExternalWritable := 'False'} : Bool;
   // END_VAR
BEGIN
END_DATA_BLOCK

DATA_BLOCK "IEC_Timer_0_DB_123"   // DB253
{ S7_Optimized_Access := 'TRUE' }
// stored: InstanceOfName IEC_TIMER, OfSystemLibElement IEC_TIMER, OfSystemLibVersion 1.0
"IEC_TIMER"
   // VAR
   //    PT : Time;
   //    ET { ExternalWritable := 'False'} : Time;
   //    IN : Bool;
   //    Q { ExternalWritable := 'False'} : Bool;
   // END_VAR
BEGIN
END_DATA_BLOCK

DATA_BLOCK "IEC_Timer_0_DB_124"   // DB254
{ S7_Optimized_Access := 'TRUE' }
// stored: InstanceOfName IEC_TIMER, OfSystemLibElement IEC_TIMER, OfSystemLibVersion 1.0
"IEC_TIMER"
   // VAR
   //    PT : Time;
   //    ET { ExternalWritable := 'False'} : Time;
   //    IN : Bool;
   //    Q { ExternalWritable := 'False'} : Bool;
   // END_VAR
BEGIN
END_DATA_BLOCK

DATA_BLOCK "IEC_Timer_0_DB_125"   // DB255
{ S7_Optimized_Access := 'TRUE' }
// stored: InstanceOfName IEC_TIMER, OfSystemLibElement IEC_TIMER, OfSystemLibVersion 1.0
"IEC_TIMER"
   // VAR
   //    PT : Time;
   //    ET { ExternalWritable := 'False'} : Time;
   //    IN : Bool;
   //    Q { ExternalWritable := 'False'} : Bool;
   // END_VAR
BEGIN
END_DATA_BLOCK

DATA_BLOCK "IEC_Timer_0_DB_126"   // DB256
{ S7_Optimized_Access := 'TRUE' }
// stored: InstanceOfName IEC_TIMER, OfSystemLibElement IEC_TIMER, OfSystemLibVersion 1.0
"IEC_TIMER"
   // VAR
   //    PT : Time;
   //    ET { ExternalWritable := 'False'} : Time;
   //    IN : Bool;
   //    Q { ExternalWritable := 'False'} : Bool;
   // END_VAR
BEGIN
END_DATA_BLOCK

DATA_BLOCK "IEC_Timer_0_DB_127"   // DB257
{ S7_Optimized_Access := 'TRUE' }
// stored: InstanceOfName IEC_TIMER, OfSystemLibElement IEC_TIMER, OfSystemLibVersion 1.0
"IEC_TIMER"
   // VAR
   //    PT : Time;
   //    ET { ExternalWritable := 'False'} : Time;
   //    IN : Bool;
   //    Q { ExternalWritable := 'False'} : Bool;
   // END_VAR
BEGIN
END_DATA_BLOCK

DATA_BLOCK "IEC_Timer_0_DB_128"   // DB258
{ S7_Optimized_Access := 'TRUE' }
// stored: InstanceOfName IEC_TIMER, OfSystemLibElement IEC_TIMER, OfSystemLibVersion 1.0
"IEC_TIMER"
   // VAR
   //    PT : Time;
   //    ET { ExternalWritable := 'False'} : Time;
   //    IN : Bool;
   //    Q { ExternalWritable := 'False'} : Bool;
   // END_VAR
BEGIN
END_DATA_BLOCK

DATA_BLOCK "IEC_Timer_0_DB_129"   // DB259
{ S7_Optimized_Access := 'TRUE' }
// stored: InstanceOfName IEC_TIMER, OfSystemLibElement IEC_TIMER, OfSystemLibVersion 1.0
"IEC_TIMER"
   // VAR
   //    PT : Time;
   //    ET { ExternalWritable := 'False'} : Time;
   //    IN : Bool;
   //    Q { ExternalWritable := 'False'} : Bool;
   // END_VAR
BEGIN
END_DATA_BLOCK

DATA_BLOCK "IEC_Timer_0_DB_13"   // DB105
{ S7_Optimized_Access := 'TRUE' }
// stored: InstanceOfName IEC_TIMER, OfSystemLibElement IEC_TIMER, OfSystemLibVersion 1.0
"IEC_TIMER"
   // VAR
   //    PT : Time;
   //    ET { ExternalWritable := 'False'} : Time;
   //    IN : Bool;
   //    Q { ExternalWritable := 'False'} : Bool;
   // END_VAR
BEGIN
END_DATA_BLOCK

DATA_BLOCK "IEC_Timer_0_DB_130"   // DB260
{ S7_Optimized_Access := 'TRUE' }
// stored: InstanceOfName IEC_TIMER, OfSystemLibElement IEC_TIMER, OfSystemLibVersion 1.0
"IEC_TIMER"
   // VAR
   //    PT : Time;
   //    ET { ExternalWritable := 'False'} : Time;
   //    IN : Bool;
   //    Q { ExternalWritable := 'False'} : Bool;
   // END_VAR
BEGIN
END_DATA_BLOCK

DATA_BLOCK "IEC_Timer_0_DB_131"   // DB261
{ S7_Optimized_Access := 'TRUE' }
// stored: InstanceOfName IEC_TIMER, OfSystemLibElement IEC_TIMER, OfSystemLibVersion 1.0
"IEC_TIMER"
   // VAR
   //    PT : Time;
   //    ET { ExternalWritable := 'False'} : Time;
   //    IN : Bool;
   //    Q { ExternalWritable := 'False'} : Bool;
   // END_VAR
BEGIN
END_DATA_BLOCK

DATA_BLOCK "IEC_Timer_0_DB_132"   // DB262
{ S7_Optimized_Access := 'TRUE' }
// stored: InstanceOfName IEC_TIMER, OfSystemLibElement IEC_TIMER, OfSystemLibVersion 1.0
"IEC_TIMER"
   // VAR
   //    PT : Time;
   //    ET { ExternalWritable := 'False'} : Time;
   //    IN : Bool;
   //    Q { ExternalWritable := 'False'} : Bool;
   // END_VAR
BEGIN
END_DATA_BLOCK

DATA_BLOCK "IEC_Timer_0_DB_133"   // DB263
{ S7_Optimized_Access := 'TRUE' }
// stored: InstanceOfName IEC_TIMER, OfSystemLibElement IEC_TIMER, OfSystemLibVersion 1.0
"IEC_TIMER"
   // VAR
   //    PT : Time;
   //    ET { ExternalWritable := 'False'} : Time;
   //    IN : Bool;
   //    Q { ExternalWritable := 'False'} : Bool;
   // END_VAR
BEGIN
END_DATA_BLOCK

DATA_BLOCK "IEC_Timer_0_DB_134"   // DB264
{ S7_Optimized_Access := 'TRUE' }
// stored: InstanceOfName IEC_TIMER, OfSystemLibElement IEC_TIMER, OfSystemLibVersion 1.0
"IEC_TIMER"
   // VAR
   //    PT : Time;
   //    ET { ExternalWritable := 'False'} : Time;
   //    IN : Bool;
   //    Q { ExternalWritable := 'False'} : Bool;
   // END_VAR
BEGIN
END_DATA_BLOCK

DATA_BLOCK "IEC_Timer_0_DB_135"   // DB265
{ S7_Optimized_Access := 'TRUE' }
// stored: InstanceOfName IEC_TIMER, OfSystemLibElement IEC_TIMER, OfSystemLibVersion 1.0
"IEC_TIMER"
   // VAR
   //    PT : Time;
   //    ET { ExternalWritable := 'False'} : Time;
   //    IN : Bool;
   //    Q { ExternalWritable := 'False'} : Bool;
   // END_VAR
BEGIN
END_DATA_BLOCK

DATA_BLOCK "IEC_Timer_0_DB_136"   // DB266
{ S7_Optimized_Access := 'TRUE' }
// stored: InstanceOfName IEC_TIMER, OfSystemLibElement IEC_TIMER, OfSystemLibVersion 1.0
"IEC_TIMER"
   // VAR
   //    PT : Time;
   //    ET { ExternalWritable := 'False'} : Time;
   //    IN : Bool;
   //    Q { ExternalWritable := 'False'} : Bool;
   // END_VAR
BEGIN
END_DATA_BLOCK

DATA_BLOCK "IEC_Timer_0_DB_137"   // DB267
{ S7_Optimized_Access := 'TRUE' }
// stored: InstanceOfName IEC_TIMER, OfSystemLibElement IEC_TIMER, OfSystemLibVersion 1.0
"IEC_TIMER"
   // VAR
   //    PT : Time;
   //    ET { ExternalWritable := 'False'} : Time;
   //    IN : Bool;
   //    Q { ExternalWritable := 'False'} : Bool;
   // END_VAR
BEGIN
END_DATA_BLOCK

DATA_BLOCK "IEC_Timer_0_DB_138"   // DB268
{ S7_Optimized_Access := 'TRUE' }
// stored: InstanceOfName IEC_TIMER, OfSystemLibElement IEC_TIMER, OfSystemLibVersion 1.0
"IEC_TIMER"
   // VAR
   //    PT : Time;
   //    ET { ExternalWritable := 'False'} : Time;
   //    IN : Bool;
   //    Q { ExternalWritable := 'False'} : Bool;
   // END_VAR
BEGIN
END_DATA_BLOCK

